# B&R Automation Studio project mappFramework (part 7)

#### HMIActions.st
```iecst
ACTION ReportFormat:

	// If the current format and the selected format do not match, disable the function block for a cycle and make the change
	IF HmiReport.Parameters.UseAdvancedFormat AND (HmiReport.Status.CurrentFormat = FORMAT_SIMPLE) THEN
		MpReportCoreSys.Enable := FALSE;
		MpReportCoreSys.MpLink := ADR(gMpLinkAdvancedReport);
		HmiReport.Parameters.Name := 'AdvancedReport';
		HmiReport.Status.CurrentFormat := FORMAT_ADVANCED;
	ELSIF NOT HmiReport.Parameters.UseAdvancedFormat AND (HmiReport.Status.CurrentFormat = FORMAT_ADVANCED) THEN
		MpReportCoreSys.Enable := FALSE;
		MpReportCoreSys.MpLink := ADR(gMpLinkSimpleReport);
		HmiReport.Parameters.Name := 'SimpleReport';
		HmiReport.Status.CurrentFormat := FORMAT_SIMPLE;
	ELSE
		MpReportCoreSys.Enable := TRUE;
	END_IF

END_ACTION

ACTION ReportFileExplorer:

	// Connections between the HMI structure and the report function block
	HmiReport.Status.Busy := MpReportCoreSys.CommandBusy;
	HmiReport.Status.Error := MpReportCoreSys.Error;
	MpReportCoreSys.Language := ADR(HmiReport.Parameters.SelectedLanguage);

	// Set or reset bits based on when a report can be created, deleted, and/or viewed.
	HmiReport.Status.CreateAllowed := NOT(MpReportCoreSys.CommandBusy);
	HmiReport.Status.ViewAllowed := (MpFileManagerUIConnect.File.List.Items[HmiReport.Status.SelectedIndex].ItemType = mpFILE_ITEM_TYPE_USER1);
	HmiReport.Status.DeleteAllowed := (MpFileManagerUIConnect.File.List.Items[HmiReport.Status.SelectedIndex].ItemType = mpFILE_ITEM_TYPE_USER1);

	// If the selected index on screen matches the index of a given file, mark that file as selected in the UIConnect structure
	FOR i := 0 TO ((SIZEOF(HmiReport.Status.FileNames)/SIZEOF(HmiReport.Status.FileNames[0])) - 1) DO
		IF (i = HmiReport.Status.SelectedIndex) AND NOT MpFileManagerUIConnect.File.List.Items[i].IsSelected THEN
			MpFileManagerUIConnect.File.List.Items[i].IsSelected := TRUE;
		ELSIF (i <> HmiReport.Status.SelectedIndex) AND MpFileManagerUIConnect.File.List.Items[i].IsSelected THEN
			MpFileManagerUIConnect.File.List.Items[i].IsSelected := FALSE;
		END_IF
	END_FOR

	// For every file, record its name, timestamp, size, and path
	FOR i := 0 TO ((SIZEOF(HmiReport.Status.FileNames)/SIZEOF(HmiReport.Status.FileNames[0])) - 1) DO
		HmiReport.Status.FileNames[i] := MpFileManagerUIConnect.File.List.Items[i].Name;
		HmiReport.Status.TimeStamps[i] := MpFileManagerUIConnect.File.List.Items[i].LastModified;

		IF MpFileManagerUIConnect.File.List.Items[i].Size <> 0 THEN
			HmiReport.Status.TimeStampsText[i] := DT_TO_STRING(MpFileManagerUIConnect.File.List.Items[i].LastModified);
			HmiReport.Status.TimeStampsText[i] := RIGHT(HmiReport.Status.TimeStampsText[i], 19);
		ELSE
			HmiReport.Status.TimeStampsText[i] := '';
		END_IF;

		HmiReport.Status.Size[i] := MpFileManagerUIConnect.File.List.Items[i].Size;
		// Concatonate strings to form the file path
		HmiReport.Status.TempFilePath[i] := '/FileDevice:';
		brsstrcat(ADR(HmiReport.Status.TempFilePath[i]),ADR(MpFileManagerUIConnect.DeviceList.DeviceNames[MpFileManagerUIConnect.DeviceList.SelectedIndex]));
		brsstrcat(ADR(HmiReport.Status.TempFilePath[i]),ADR('/'));
		brsstrcat(ADR(HmiReport.Status.TempFilePath[i]),ADR(HmiReport.Status.FileNames[i]));
		HmiReport.Status.FilePath[i] := HmiReport.Status.TempFilePath[i];
	END_FOR

	// Create a file path to be linked to the pdf viewer
	HmiReport.Parameters.PathOfReportToView := HmiReport.Status.FilePath[HmiReport.Status.SelectedIndex];

	// Add USB devices if available
	FOR i := 0 TO IDX_USB_DEV_LIST DO
		tempDeviceIndex := i + 1;
		IF gUSBAvailable[i] THEN
			MpFileManagerUIConnect.DeviceList.DeviceNames[tempDeviceIndex] := 'USB';
			brsitoa(i + 1, ADR(MpFileManagerUIConnect.DeviceList.DeviceNames[tempDeviceIndex]) + brsstrlen(ADR(MpFileManagerUIConnect.DeviceList.DeviceNames[tempDeviceIndex])));
		ELSE
			MpFileManagerUIConnect.DeviceList.DeviceNames[tempDeviceIndex] := '';
		END_IF
	END_FOR

	// Create array for the file device table
	IF ((MpFileManagerUIConnect.DeviceList.SelectedIndex <> HmiReport.Status.LastSelectedDeviceIndex) AND (MpFileManagerUIConnect.Status = mpFILE_UI_STATUS_IDLE)) THEN
		HmiReport.Status.LastSelectedDeviceIndex := MpFileManagerUIConnect.DeviceList.SelectedIndex;
		HmiReport.Status.LastSelectedIndex := HmiReport.Status.LastSelectedIndex + 1;
	END_IF

	// If more than 50 items exist, set the File OverMax flag (used for page up/down buttons)
	HmiReport.Status.FileOverMax := ItemCount > 50;

	// Set file device to selected
	MpReportCoreSys.DeviceName := ADR(MpFileManagerUIConnect.DeviceList.DeviceNames[MpFileManagerUIConnect.DeviceList.SelectedIndex]);

	// VC4
	IF HmiReport.Status.Error THEN
		HmiReport.Status.Layer.ReportCreate := USINT_TO_BOOL(HIDE);
	END_IF
	IF HmiReport.Status.DeleteAllowed THEN
		HmiReport.Status.DeleteButtonEnableStatus := USINT_TO_BOOL(HIDE);
	ELSE
		HmiReport.Status.DeleteButtonEnableStatus := USINT_TO_BOOL(DISPLAY);
	END_IF
	IF HmiReport.Status.FileOverMax THEN
		HmiReport.Status.PageUpDownVisibility := DISPLAY;
	ELSE
		HmiReport.Status.PageUpDownVisibility := HIDE;
	END_IF

	// Language assignments
	CASE HmiReport.Parameters.Language OF

		// English
		0:
			MpReportCoreSys.Language := ADR('en');
		// German
		1:
			MpReportCoreSys.Language := ADR('de');
		// Chinese
		2:
			MpReportCoreSys.Language := ADR('zh');

	END_CASE

END_ACTION
```

#### ReportMgr.st
```iecst
//***********************************************************************
// Copyright: B&R Industrial Automation GmbH
// Author: B&R Industrial Automation GmbH
// Created: Dec 1, 2022
// Description: Task for generating reports with VC4 front-end.
//***********************************************************************

PROGRAM _INIT

	// Create folder for this component on the user file device
	DirCreateReport(enable := TRUE, pDevice := ADR('mappReportFiles'), pName := ADR('/'));

	// Check if folder already exist and if so disabled the function block call
	IF DirCreateReport.status = fiERR_DIR_ALREADY_EXIST THEN
		DirCreateReport(enable := FALSE);
	END_IF

	// Initialize mapp function blocks
	MpReportCoreSys.Language := ADR('en');
	MpReportCoreSys.DeviceName := ADR('mappReportFiles');
	MpReportCoreSys.MpLink := ADR(gMpLinkSimpleReport);
	MpReportCoreSys.Name := ADR(HmiReport.Parameters.Name);
	HmiReport.Parameters.Name := 'SimpleReport';
	HmiReport.Parameters.SortType := 'NameAsc';
	MpReportCoreSys();

	MpFileManagerUIReport.MpLink := ADR(gMpLinkFileManagerUIReport);
	MpFileManagerUIReport.UIConnect := ADR(MpFileManagerUIConnect);
	MpFileManagerUIReport.UISetup.FileListSize := SIZEOF(MpFileManagerUIConnect.File.List.Items) / SIZEOF(MpFileManagerUIConnect.File.List.Items[0]);
	MpFileManagerUIReport.Enable := TRUE;
	MpFileManagerUIReport();

	// Fill an array to create example data for the example report
	TimeIndex := 0;
	FOR i:=0 TO ((SIZEOF(ReportExample.SimpleReport.OeeLine[0].TemperatureSample.TimeStamp)/SIZEOF(ReportExample.SimpleReport.OeeLine[0].TemperatureSample.TimeStamp[0])) - 1) DO
		ReportExample.SimpleReport.OeeLine[0].TemperatureSample.TimeStamp[i] := TimeIndex;
		ReportExample.SimpleReport.OeeLine[1].TemperatureSample.TimeStamp[i] := TimeIndex;
		ReportExample.SimpleReport.OeeLine[2].TemperatureSample.TimeStamp[i] := TimeIndex;
		ReportExample.AdvancedReport.OeeLine[0].TemperatureSample.TimeStamp[i] := TimeIndex;
		ReportExample.AdvancedReport.OeeLine[1].TemperatureSample.TimeStamp[i] := TimeIndex;
		ReportExample.AdvancedReport.OeeLine[2].TemperatureSample.TimeStamp[i] := TimeIndex;
		TimeIndex := TimeIndex + 15;
	END_FOR

	// Ficticious number to serve as an example in the report
	ReportExample.AdvancedReport.BatchNumber := 325454685;

END_PROGRAM

PROGRAM _CYCLIC

	// Once a report has been generated, clear the generate command
	IF MpReportCoreSys.CommandDone THEN
		MpFileManagerUIConnect.File.Refresh := TRUE;
		HmiReport.Commands.Generate := FALSE;
	END_IF

	// Call all cyclic actions
	ReportFormat;
	ReportFileExplorer;

	// Generate command
	MpReportCoreSys.Generate := HmiReport.Commands.Generate;
	MpReportCoreSys.Name := ADR(HmiReport.Parameters.Name);

	// Assign address references
	MpFileManagerUIReport.UIConnect := ADR(MpFileManagerUIConnect);
	MpFileManagerUIReport.MpLink := ADR(gMpLinkFileManagerUIReport);
	MpFileManagerUIReport.UIConnect := ADR(MpFileManagerUIConnect);

	// Call function blocks
	MpReportCoreSys();
	MpFileManagerUIReport();

END_PROGRAM

PROGRAM _EXIT

	// Disable the function blocks to unlink the MpLinks
	MpReportCoreSys.Enable := FALSE;
	MpFileManagerUIReport.Enable := FALSE;

	// Call function blocks
	MpReportCoreSys();
	MpFileManagerUIReport();

END_PROGRAM
```

### mappFrameworkVC4.var - not listed in the package file held
```iecst
(*Constants*)
VAR CONSTANT
	DISPLAY : USINT := 0; (*VC4 visibility control*)
	HIDE : USINT := 1; (*VC4 visibility control*)
	OPERATION_ACTIVATED : USINT := 1; (*VC4 access control*)
	OPERATION_DEACTIVATED : USINT := 0; (*VC4 access control*)
	LOCK : USINT := 0; (*VC4 lock control*)
	UNLOCK : USINT := 1; (*VC4 unlock control*)
END_VAR
```

### Program Logical/Infrastructure/VC4/PackML/PackMLMgr (IEC)

#### PackMLMgr.st - Init, cyclic, exit code
```iecst
//***********************************************************************
// Copyright: B&R Industrial Automation GmbH
// Author: B&R Industrial Automation GmbH
// Created: June 1, 2023
// Description: Task for handling PackML control with VC4 front-end.
//***********************************************************************

PROGRAM _INIT

	// NOTE: For VC4 implementations, the MpPackMLCore must be configured in "standalone" mode.
	// For additional information, see "Required Modifications" in AS Mapp Framework Help.

	// Create folder for this component on the user file device
	DirCreatePackML(enable := TRUE, pDevice := ADR('mappPackMLFiles'), pName := ADR('/'));

	// Check if folder already exist and if so disabled the function block call
	IF DirCreatePackML.status = fiERR_DIR_ALREADY_EXIST THEN
		DirCreatePackML(enable := FALSE);
	END_IF

	// Initialize mapp function blocks
	MpPackMLCoreMain.MpLink := ADR(gMpLinkPackMLCore);
	MpPackMLCoreMain.Enable := TRUE;
	MpPackMLCoreMain();

	MpPackMLModeMain.MpLink := ADR(gMpLinkPackMLCore);
	MpPackMLModeMain.Enable := TRUE;
	MpPackMLModeMain.ModeID := 1;
	MpPackMLModeMain();

	MpPackMLBasicUIMain.MpLink := ADR(gMpLinkPackMLCore);
	MpPackMLBasicUIMain.Enable := TRUE;
	MpPackMLBasicUIMain.UIConnect := ADR(MpPackMLBasicUIConnect);
	MpPackMLBasicUIMain();

	MpPackMLStatisticsUIMain.MpLink := ADR(gMpLinkPackMLCore);
	MpPackMLStatisticsUIMain.Enable := TRUE;
	MpPackMLStatisticsUIMain.UIConnect := ADR(MpPackMLStatisticsUIConnect);
	MpPackMLStatisticsUIMain();

	// Assign Production mode as selected Index since it's the start mode and preselected
	MpPackMLBasicUIConnect.ModeControl.SelectedIndex := 1;

END_PROGRAM

PROGRAM _CYCLIC

	// Call all cyclic actions
	StateMachine;

	// Assign MpLinks & UIConnects
	MpPackMLCoreMain.MpLink := ADR(gMpLinkPackMLCore);
	MpPackMLModeMain.MpLink := ADR(gMpLinkPackMLCore);
	MpPackMLBasicUIMain.MpLink := ADR(gMpLinkPackMLCore);
	MpPackMLStatisticsUIMain.MpLink := ADR(gMpLinkPackMLCore);

	// Call function blocks
	MpPackMLCoreMain();
	MpPackMLModeMain();
	MpPackMLBasicUIMain();
	MpPackMLStatisticsUIMain();

END_PROGRAM

PROGRAM _EXIT

	// Disable the function blocks to unlink the MpLinks
	MpPackMLCoreMain.Enable := FALSE;
	MpPackMLModeMain.Enable := FALSE;
	MpPackMLBasicUIMain.Enable := FALSE;
	MpPackMLStatisticsUIMain.Enable := TRUE;

	// Call function blocks
	MpPackMLCoreMain();
	MpPackMLModeMain();
	MpPackMLBasicUIMain();
	MpPackMLStatisticsUIMain();

END_PROGRAM
```

#### PackMLMgr.var - Local variables
```iecst
(*Function Blocks*)
VAR
	DirCreatePackML : DirCreate; (*DirCreate instance*)
	MpPackMLCoreMain : MpPackMLCore;
	MpPackMLModeMain : MpPackMLMode;
	MpPackMLBasicUIMain : MpPackMLBasicUI;
	MpPackMLStatisticsUIMain : MpPackMLStatisticsUI;
END_VAR
(*Constants*)
(*Structure Types*)
VAR
	MpPackMLBasicUIConnect : MpPackMLBasicUIConnectType;
END_VAR
(*Variables*)
VAR
	MpPackMLStatisticsUIConnect : MpPackMLStatisticsUIConnectType;
END_VAR
```

#### StateMachine.st
```iecst
ACTION StateMachine:

	CASE MpPackMLCoreMain.StateCurrent OF

		mpPACKML_STATE_STOPPED:

			// Add STOPPED actions here
			MpPackMLModeMain.StateComplete := FALSE;

		mpPACKML_STATE_STARTING:

			// Add STARTING actions here
			MpPackMLModeMain.StateComplete := TRUE;

		mpPACKML_STATE_IDLE:

			// Add IDLE actions here
			MpPackMLModeMain.StateComplete := FALSE;

		mpPACKML_STATE_SUSPENDING:

			// Add SUSPENDING actions here
			MpPackMLModeMain.StateComplete := TRUE;

		mpPACKML_STATE_SUSPENDED:

			// Add SUSPENDED actions here
			MpPackMLModeMain.StateComplete := FALSE;

		mpPACKML_STATE_UNSUSPENDING:

			// Add UNSUSPENDING actions here
			MpPackMLModeMain.StateComplete := TRUE;

		mpPACKML_STATE_EXECUTE:

			// Add EXECUTE actions here
			MpPackMLModeMain.StateComplete := FALSE;

		mpPACKML_STATE_STOPPING:

			// Add STOPPING actions here
			MpPackMLModeMain.StateComplete := TRUE;

		mpPACKML_STATE_ABORTING:

			// Add ABORTING actions here
			MpPackMLModeMain.StateComplete := TRUE;

		mpPACKML_STATE_ABORTED:

			// Add ABORTED actions here
			MpPackMLModeMain.StateComplete := FALSE;

		mpPACKML_STATE_HOLDING:

			// Add HOLDING actions here
			MpPackMLModeMain.StateComplete := TRUE;

		mpPACKML_STATE_HELD:

			// Add HELD actions here
			MpPackMLModeMain.StateComplete := FALSE;

		mpPACKML_STATE_UNHOLDING:

			// Add UNHOLDING actions here
			MpPackMLModeMain.StateComplete := TRUE;

		mpPACKML_STATE_COMPLETING:

			// Add COMPLETING actions here
			MpPackMLModeMain.StateComplete := TRUE;

			// NOTE: To allow the state machine to move forward, the StateComplete command has been connected
			// to the HMI button. The user should change this to set StateComplete to TRUE upon COMPLETING actions.

		mpPACKML_STATE_COMPLETE:

			// Add COMPLETE actions here
			MpPackMLModeMain.StateComplete := FALSE;

		mpPACKML_STATE_RESETTING:

			// Add RESETTING actions here
			MpPackMLModeMain.StateComplete := TRUE;

		mpPACKML_STATE_CLEARING:

			// Add CLEARING actions here
			MpPackMLModeMain.StateComplete := TRUE;

		mpPACKML_STATE_UNDEFINED:

			// Add UNDEFINED actions here
			MpPackMLModeMain.Activate := TRUE;

		mpPACKML_STATE_DEACTIVATING:

			// Add DEACTIVATING actions here

		mpPACKML_STATE_DEACTIVATED:

			// Add DEACTIVATED actions here

		mpPACKML_STATE_ACTIVATING:

			// Add ACTIVATING actions here

			MpPackMLModeMain.StateComplete := TRUE;

	END_CASE

END_ACTION
```

#### HMIActions.st - not listed in the package file held
```iecst
ACTION VC4_Cyclic:

	IF HmiPackML.Status.LastState <> MpPackMLMode_0.StateCurrent THEN

		// Reset all commands on each state change
		MpPackMLBasicUIConnect.StateControl.Abort := MpPackMLMode_0.Abort := FALSE;
		MpPackMLBasicUIConnect.StateControl.Clear := MpPackMLMode_0.Clear := FALSE;
		MpPackMLBasicUIConnect.StateControl.Hold := MpPackMLMode_0.Hold := FALSE;
		MpPackMLBasicUIConnect.StateControl.Reset := MpPackMLMode_0.Reset := FALSE;
		MpPackMLBasicUIConnect.StateControl.Start := MpPackMLMode_0.Start := FALSE;
		MpPackMLBasicUIConnect.StateControl.StateComplete := MpPackMLMode_0.StateComplete := FALSE;
		MpPackMLBasicUIConnect.StateControl.Stop := MpPackMLMode_0.Stop := FALSE;
		MpPackMLBasicUIConnect.StateControl.Suspend := MpPackMLMode_0.Suspend := FALSE;
		MpPackMLBasicUIConnect.StateControl.Unhold := MpPackMLMode_0.Unhold := FALSE;
		MpPackMLBasicUIConnect.StateControl.Unsuspend := MpPackMLMode_0.Unsuspend := FALSE;

		// Reset all ColorIndexes on each state change
		MpPackMLBasicUIConnect.StateControl.ColorIndex.Stopped := 0;
		MpPackMLBasicUIConnect.StateControl.ColorIndex.Stopping := 0;
		MpPackMLBasicUIConnect.StateControl.ColorIndex.Clearing := 0;
		MpPackMLBasicUIConnect.StateControl.ColorIndex.Aborted := 0;
		MpPackMLBasicUIConnect.StateControl.ColorIndex.Aborting := 0;
		MpPackMLBasicUIConnect.StateControl.ColorIndex.Resetting := 0;
		MpPackMLBasicUIConnect.StateControl.ColorIndex.Unsuspending := 0;
		MpPackMLBasicUIConnect.StateControl.ColorIndex.Suspended := 0;
		MpPackMLBasicUIConnect.StateControl.ColorIndex.Suspending := 0;
		MpPackMLBasicUIConnect.StateControl.ColorIndex.Idle := 0;
		MpPackMLBasicUIConnect.StateControl.ColorIndex.Starting := 0;
		MpPackMLBasicUIConnect.StateControl.ColorIndex.Execute := 0;
		MpPackMLBasicUIConnect.StateControl.ColorIndex.Completing := 0;
		MpPackMLBasicUIConnect.StateControl.ColorIndex.Complete := 0;
		MpPackMLBasicUIConnect.StateControl.ColorIndex.Unholding := 0;
		MpPackMLBasicUIConnect.StateControl.ColorIndex.Held := 0;
		MpPackMLBasicUIConnect.StateControl.ColorIndex.Holding := 0;

		HmiPackML.Status.LastState := MpPackMLMode_0.StateCurrent;

	END_IF

	// Connect UIConnect Commands to function block
	MpPackMLMode_0.Abort := MpPackMLBasicUIConnect.StateControl.Abort;
	MpPackMLMode_0.Stop := MpPackMLBasicUIConnect.StateControl.Stop;

	MpPackMLBasicUIConnect.ModeCurrent := MpPackMLMode_0.ModeID;
	MpPackMLBasicUIConnect.StateCurrent := MpPackMLMode_0.StateCurrent;

END_ACTION
```

#### StateMachine_Main.st - not listed in the package file held
```iecst
ACTION StateMachine_Main:

	CASE MpPackMLCore_0.StateCurrent OF

		mpPACKML_STATE_STOPPED:

			// Add STOPPED actions here
			MpPackMLMode_0.StateComplete := FALSE;

		mpPACKML_STATE_STARTING:

			// Add STARTING actions here
			MpPackMLMode_0.StateComplete := TRUE;

		mpPACKML_STATE_IDLE:

			// Add IDLE actions here
			MpPackMLMode_0.StateComplete := FALSE;

		mpPACKML_STATE_SUSPENDING:

			// Add SUSPENDING actions here
			MpPackMLMode_0.StateComplete := TRUE;

		mpPACKML_STATE_SUSPENDED:

			// Add SUSPENDED actions here
			MpPackMLMode_0.StateComplete := FALSE;

		mpPACKML_STATE_UNSUSPENDING:

			// Add UNSUSPENDING actions here
			MpPackMLMode_0.StateComplete := TRUE;

		mpPACKML_STATE_EXECUTE:

			// Add EXECUTE actions here
			MpPackMLMode_0.StateComplete := FALSE;

		mpPACKML_STATE_STOPPING:

			// Add STOPPING actions here
			MpPackMLMode_0.StateComplete := TRUE;

		mpPACKML_STATE_ABORTING:

			// Add ABORTING actions here
			MpPackMLMode_0.StateComplete := TRUE;

		mpPACKML_STATE_ABORTED:

			// Add ABORTED actions here
			MpPackMLMode_0.StateComplete := FALSE;

		mpPACKML_STATE_HOLDING:

			// Add HOLDING actions here
			MpPackMLMode_0.StateComplete := TRUE;

		mpPACKML_STATE_HELD:

			// Add HELD actions here
			MpPackMLMode_0.StateComplete := FALSE;

		mpPACKML_STATE_UNHOLDING:

			// Add UNHOLDING actions here
			MpPackMLMode_0.StateComplete := TRUE;

		mpPACKML_STATE_COMPLETING:

			// Add COMPLETING actions here
			MpPackMLMode_0.StateComplete := TRUE;

			// NOTE: To allow the state machine to move forward, the StateComplete command has been connected
			// to the HMI button. The user should change this to set StateComplete to TRUE upon COMPLETING actions.

		mpPACKML_STATE_COMPLETE:

			// Add COMPLETE actions here
			MpPackMLMode_0.StateComplete := FALSE;

		mpPACKML_STATE_RESETTING:

			// Add RESETTING actions here
			MpPackMLMode_0.StateComplete := TRUE;

		mpPACKML_STATE_CLEARING:

			// Add CLEARING actions here
			MpPackMLMode_0.StateComplete := TRUE;

		mpPACKML_STATE_UNDEFINED:

			// Add UNDEFINED actions here
			MpPackMLMode_0.Activate := TRUE;

		mpPACKML_STATE_DEACTIVATING:

			// Add DEACTIVATING actions here

		mpPACKML_STATE_DEACTIVATED:

			// Add DEACTIVATED actions here

		mpPACKML_STATE_ACTIVATING:

			// Add ACTIVATING actions here

			MpPackMLMode_0.StateComplete := TRUE;

	END_CASE

END_ACTION
```

### Program Logical/Infrastructure/PackML/PackMLMgr (IEC) - Pack ML Manager

#### PackMLMgr.st - Init, cyclic, exit code
```iecst
//***********************************************************************
// Copyright: B&R Industrial Automation GmbH
// Author: B&R Industrial Automation GmbH
// Created: June 1, 2023
// Description: Task for handling PackML control.
//***********************************************************************

PROGRAM _INIT

	// Create folder for this component on the user file device
	DirCreatePackML(enable := TRUE, pDevice := ADR('mappPackMLFiles'), pName := ADR('/'));

	// Check if folder already exist and if so disabled the function block call
	IF DirCreatePackML.status = fiERR_DIR_ALREADY_EXIST THEN
		DirCreatePackML(enable := FALSE);
	END_IF

	// Initialize mapp function blocks
	MpPackMLModuleMain.Parameters := ADR(MpPackMLModuleParMain);
	MpPackMLModuleMain.MpLink := ADR(gMpPackMLModuleMain);
	MpPackMLModuleMain.Enable := TRUE;
	MpPackMLModuleMain();

	//PackML Mode Initializations
	StateInitialize;

	// Initialize startup mode - Automatic Mode
	HmiPackML.Commands.Mode := 1;

END_PROGRAM

PROGRAM _CYCLIC

	// Call all cyclic actions
	StateMachine;
	HmiActions;

	// Assign MpLinks & UIConnects
	MpPackMLModuleMain.Parameters := ADR(MpPackMLModuleParMain);
	MpPackMLModuleMain.MpLink := ADR(gMpPackMLModuleMain);

	// Call function blocks
	MpPackMLModuleMain();

END_PROGRAM

PROGRAM _EXIT

	// Disable the function blocks to unlink the MpLinks
	MpPackMLModuleMain.Enable := FALSE;

	// Call function blocks
	MpPackMLModuleMain();

END_PROGRAM
```

#### PackMLMgr.typ - Local data types
```iecst
(*Structure types*)

TYPE
	PackMLHmiInterfaceType : 	STRUCT  (*Structure to hold commands, parameters and status from the HMI*)
		Commands : PackMLCommandsType;
		Parameters : PackMLParametersType;
		Status : PackMLStatusType;
		Activate : BOOL;
	END_STRUCT;
	PackMLCommandsType : 	STRUCT  (*Structure to hold the commands from the HMI*)
		Reset : BOOL;
		Start : BOOL;
		Stop : BOOL;
		Hold : BOOL;
		Unhold : BOOL;
		Suspend : BOOL;
		Unsuspend : BOOL;
		Abort : BOOL;
		Clear : BOOL;
		Complete : BOOL;
		Mode : DINT;
	END_STRUCT;
	PackMLParametersType : 	STRUCT  (*Structure to hold the parameters for the HMI*)
		Par : USINT;
		StateEnabled : PackMLStateEnabledType;
	END_STRUCT;
	PackMLStatusType : 	STRUCT  (*Structure to hold status information from the mapp View HMI*)
		StateCurrent : STRING[20];
		ModeCurrent : STRING[50];
		DownTimeReason : STRING[255];
		PackMLStateModel : STRING[100000];
		PackMLState : MpPackMLStateEnum;
	END_STRUCT;
	PackMLStateEnabledType : 	STRUCT  (*Structure to hold state availability definition*)
		Clearing : BOOL; (*Statistic information for Clearing state*)
		Stopped : BOOL; (*Statistic information for Stopped state*)
		Starting : BOOL; (*Statistic information for Starting state*)
		Idle : BOOL; (*Statistic information for Idle state*)
		Suspended : BOOL; (*Statistic information for Suspended state*)
		Execute : BOOL; (*Statistic information for Execute state*)
		Stopping : BOOL; (*Statistic information for Stopping state*)
		Aborting : BOOL; (*Statistic information for Aborting state*)
		Aborted : BOOL; (*Statistic information for Aborted state*)
		Holding : BOOL; (*Statistic information for Holding state*)
		Held : BOOL; (*Statistic information for Held state*)
		Unholding : BOOL; (*Statistic information for Unholding state*)
		Suspending : BOOL; (*Statistic information for Suspending state*)
		Unsuspending : BOOL; (*Statistic information for Unsuspending state*)
		Resetting : BOOL; (*Statistic information for Resetting state*)
		Completing : BOOL; (*Statistic information for Completing state*)
		Complete : BOOL; (*Statistic information for Complete state*)
	END_STRUCT;
END_TYPE

(*Enumerations*)
```

#### PackMLMgr.var - Local variables
```iecst
(*Function Blocks*)
VAR
	DirCreatePackML : DirCreate; (*DirCreate instance*)
	MpPackMLModuleMain : MpPackMLModule; (*PackMLModule instance*)
	MpPackMLModuleParMain : MpPackMLModuleParType; (*PackMLModule Parameter instance*)
	StateBlinkTimer : TON; (*Timer to control state blinking action*)
END_VAR
(*Constants*)
(*Structure Types*)
VAR
	Manual : PackMLStateEnabledType; (*State active / inactive control*)
	Maintenance : PackMLStateEnabledType; (*State active / inactive control*)
	AutomaticMode : PackMLStateEnabledType; (*State active / inactive control*)
	HmiPackML : PackMLHmiInterfaceType; (*HMI interface structure*)
END_VAR
(*Variables*)
```

#### HMIActions.st - Supporting code for the HMI interface
```iecst
ACTION HmiActions:

	// Connect HMIPackML Commands to function block
	MpPackMLModuleMain.Command.Abort := HmiPackML.Commands.Abort;
	MpPackMLModuleMain.Command.Clear := HmiPackML.Commands.Clear;
	MpPackMLModuleMain.Command.Hold := HmiPackML.Commands.Hold;
	MpPackMLModuleMain.Command.Reset := HmiPackML.Commands.Reset;
	MpPackMLModuleMain.Command.Start := HmiPackML.Commands.Start;
	MpPackMLModuleMain.Command.Stop := HmiPackML.Commands.Stop;
	MpPackMLModuleMain.Command.Suspend := HmiPackML.Commands.Suspend;
	MpPackMLModuleMain.Command.Unhold := HmiPackML.Commands.Unhold;
	MpPackMLModuleMain.Command.Unsuspend := HmiPackML.Commands.Unsuspend;

	// Allow user to command StateComplete only while machine is in state execute
	IF MpPackMLModuleMain.StateCurrent = mpPACKML_STATE_EXECUTE THEN
		MpPackMLModuleMain.Command.StateComplete := HmiPackML.Commands.Complete;
	END_IF

	// Assign mode configuration based on active mode
	CASE MpPackMLModuleMain.ModeID OF
		1:
			HmiPackML.Parameters.StateEnabled := AutomaticMode;
		2:
			HmiPackML.Parameters.StateEnabled := Maintenance;
		3:
			HmiPackML.Parameters.StateEnabled := Manual;
	END_CASE

	// control state machine active state blinking
	CASE HmiPackML.Status.PackMLState OF

		0:	// Build the intital string to setup enabled states and reduce the opacity to 50% for inactive states

			PackMLBaseModel(HmiPackML.Parameters.StateEnabled,ADR(HmiPackML.Status.PackMLStateModel));

			//start timer before transitioning to the current state which turns the opacity to 100% creating a blinking effect
			StateBlinkTimer.IN := TRUE;
			IF StateBlinkTimer.Q THEN
				HmiPackML.Status.PackMLState := MpPackMLModuleMain.StateCurrent;
				StateBlinkTimer.IN := FALSE;
			END_IF

		mpPACKML_STATE_CLEARING..mpPACKML_STATE_COMPLETE:

			StateBlinkTimer.IN := TRUE;
			IF StateBlinkTimer.Q THEN
				HmiPackML.Status.PackMLState := 0;
				StateBlinkTimer.IN := FALSE;
			END_IF

		ELSE	//if the state does't exist because of the synchronized mode use just go back to state 0
			HmiPackML.Status.PackMLState := 0;
	END_CASE

	// timer function block call
	StateBlinkTimer(PT := t#1s);

	// copy status info to HMI structure
	HmiPackML.Status.StateCurrent := MpPackMLModuleMain.Info.StateCurrent;
	HmiPackML.Status.ModeCurrent := MpPackMLModuleMain.Info.ModeCurrent;

END_ACTION
```

#### StateMachine.st - Main state machine logic
```iecst
ACTION StateMachine:

	// Check active state and change mode if allowed
	IF MpPackMLModeChangeIsAllowed(gMpLinkPackMLCore,HmiPackML.Commands.Mode) = 0 THEN
		MpPackMLChangeMode(gMpLinkPackMLCore,HmiPackML.Commands.Mode);
	END_IF

	CASE MpPackMLModuleMain.StateCurrent OF

		mpPACKML_STATE_STOPPED:

			// Add STOPPED actions here

		mpPACKML_STATE_STARTING:

			// Add STARTING actions here

			MpPackMLModuleMain.Command.StateComplete := TRUE;

		mpPACKML_STATE_IDLE:

			// Add IDLE actions here

		mpPACKML_STATE_SUSPENDING:

			// Add SUSPENDING actions here

			MpPackMLModuleMain.Command.StateComplete := TRUE;

		mpPACKML_STATE_SUSPENDED:

			// Add SUSPENDED actions here

		mpPACKML_STATE_UNSUSPENDING:

			// Add UNSUSPENDING actions here

			MpPackMLModuleMain.Command.StateComplete := TRUE;

		mpPACKML_STATE_EXECUTE:

			// Add EXECUTE actions here

		mpPACKML_STATE_STOPPING:

			// Add STOPPING actions here

			MpPackMLModuleMain.Command.StateComplete := TRUE;

		mpPACKML_STATE_ABORTING:

			// Add ABORTING actions here

			MpPackMLModuleMain.Command.StateComplete := TRUE;

		mpPACKML_STATE_ABORTED:

			// Add ABORTED actions here

		mpPACKML_STATE_HOLDING:

			// Add HOLDING actions here

			MpPackMLModuleMain.Command.StateComplete := TRUE;

		mpPACKML_STATE_HELD:

			// Add HELD actions here

		mpPACKML_STATE_UNHOLDING:

			// Add UNHOLDING actions here

			MpPackMLModuleMain.Command.StateComplete := TRUE;

		mpPACKML_STATE_COMPLETING:

			// Add COMPLETING actions here

			// NOTE: once COMPLETING actions that take more than one cyclic have been added, the below line
			// should be removed and replaced by the following line.
			MpPackMLModuleMain.Command.StateComplete := NOT MpPackMLModuleMain.Command.StateComplete;
			// MpPackMLModuleMain.Command.StateComplete := TRUE;

		mpPACKML_STATE_COMPLETE:

			// Add COMPLETE actions here

		mpPACKML_STATE_RESETTING:

			// Add RESETTING actions here

			MpPackMLModuleMain.Command.StateComplete := TRUE;

		mpPACKML_STATE_CLEARING:

			// Add CLEARING actions here

			MpPackMLModuleMain.Command.StateComplete := TRUE;

		mpPACKML_STATE_DEACTIVATING:

			// Add DEACTIVATING actions here

		mpPACKML_STATE_DEACTIVATED:

			// Add DEACTIVATED actions here

		mpPACKML_STATE_ACTIVATING:

			// Add ACTIVATING actions here

			MpPackMLModuleMain.Command.StateComplete := TRUE;

	END_CASE

END_ACTION
```

#### LocalFunctions.fun - Declaration for local helper functions
```iecst
{REDUND_ERROR} FUNCTION PackMLBaseModel : BOOL (* *) (*$GROUP=User,$CAT=User,$GROUPICON=User.png,$CATICON=User.png*)
	VAR_INPUT
		StateEnabled : PackMLStateEnabledType;
		BaseLayout : REFERENCE TO STRING[100000];
	END_VAR
	VAR
		stringPart : STRING[79];
	END_VAR
END_FUNCTION
```

#### PackMLBaseModel.st - Function to control the paper widget transform string
```iecst
FUNCTION PackMLBaseModel

			BaseLayout := '';
			brsstrcat(ADR(BaseLayout),ADR('['));

			IF StateEnabled.Clearing THEN
				stringPart := '{"select":"#Clearing","style":"fill:1;fill-opacity:1"}';
			ELSE
				stringPart := '{"select":"#Clearing","style":"fill:0;fill-opacity:0.5"}';
			END_IF

			brsstrcat(ADR(BaseLayout),ADR(stringPart));
			brsstrcat(ADR(BaseLayout),ADR(','));

			stringPart := '{"select":"#Stopped","style":"fill:2;fill-opacity:1"}';

			brsstrcat(ADR(BaseLayout),ADR(stringPart));
			brsstrcat(ADR(BaseLayout),ADR(','));

			IF StateEnabled.Starting THEN
				stringPart := '{"select":"#Starting","style":"fill:1;fill-opacity:1"}';
			ELSE
				stringPart := '{"select":"#Starting","style":"fill:0;fill-opacity:0.5"}';
			END_IF

			brsstrcat(ADR(BaseLayout),ADR(stringPart));
			brsstrcat(ADR(BaseLayout),ADR(','));

			stringPart := '{"select":"#Idle","style":"fill:2;fill-opacity:1"}';

			brsstrcat(ADR(BaseLayout),ADR(stringPart));
			brsstrcat(ADR(BaseLayout),ADR(','));

			IF StateEnabled.Suspended THEN
				stringPart := '{"select":"#Suspended","style":"fill:2;fill-opacity:1"}';
			ELSE
				stringPart := '{"select":"#Suspended","style":"fill:0;fill-opacity:0.5"}';
			END_IF

			brsstrcat(ADR(BaseLayout),ADR(stringPart));
			brsstrcat(ADR(BaseLayout),ADR(','));

			stringPart := '{"select":"#Execute","style":"fill:4;fill-opacity:1"}';

			brsstrcat(ADR(BaseLayout),ADR(stringPart));
			brsstrcat(ADR(BaseLayout),ADR(','));

			IF StateEnabled.Stopping THEN
				stringPart := '{"select":"#Stopping","style":"fill:1;fill-opacity:1"}';
			ELSE
				stringPart := '{"select":"#Stopping","style":"fill:0;fill-opacity:0.5"}';
			END_IF

			brsstrcat(ADR(BaseLayout),ADR(stringPart));
			brsstrcat(ADR(BaseLayout),ADR(','));

			IF StateEnabled.Aborting THEN
				stringPart := '{"select":"#Aborting","style":"fill:1;fill-opacity:1"}';
			ELSE
				stringPart := '{"select":"#Aborting","style":"fill:0;fill-opacity:0.5"}';
			END_IF

			brsstrcat(ADR(BaseLayout),ADR(stringPart));
			brsstrcat(ADR(BaseLayout),ADR(','));

			stringPart := '{"select":"#Aborted","style":"fill:2;fill-opacity:1"}';

			brsstrcat(ADR(BaseLayout),ADR(stringPart));
			brsstrcat(ADR(BaseLayout),ADR(','));

			IF StateEnabled.Holding THEN
				stringPart := '{"select":"#Holding","style":"fill:1;fill-opacity:1"}';
			ELSE
				stringPart := '{"select":"#Holding","style":"fill:0;fill-opacity:0.5"}';
			END_IF

			brsstrcat(ADR(BaseLayout),ADR(stringPart));
			brsstrcat(ADR(BaseLayout),ADR(','));

			IF StateEnabled.Held THEN
				stringPart := '{"select":"#Held","style":"fill:2;fill-opacity:1"}';
			ELSE
				stringPart := '{"select":"#Held","style":"fill:0;fill-opacity:0.5"}';
			END_IF

			brsstrcat(ADR(BaseLayout),ADR(stringPart));
			brsstrcat(ADR(BaseLayout),ADR(','));

			IF StateEnabled.Unholding THEN
				stringPart := '{"select":"#Unholding","style":"fill:1;fill-opacity:1"}';
			ELSE
				stringPart := '{"select":"#Unholding","style":"fill:0;fill-opacity:0.5"}';
			END_IF

			brsstrcat(ADR(BaseLayout),ADR(stringPart));
			brsstrcat(ADR(BaseLayout),ADR(','));

			IF StateEnabled.Suspending THEN
				stringPart := '{"select":"#Suspending","style":"fill:1;fill-opacity:1"}';
			ELSE
				stringPart := '{"select":"#Suspending","style":"fill:0;fill-opacity:0.5"}';
			END_IF

			brsstrcat(ADR(BaseLayout),ADR(stringPart));
			brsstrcat(ADR(BaseLayout),ADR(','));

			IF StateEnabled.Unsuspending THEN
				stringPart := '{"select":"#Unsuspending","style":"fill:1;fill-opacity:1"}';
			ELSE
				stringPart := '{"select":"#Unsuspending","style":"fill:0;fill-opacity:0.5"}';
			END_IF

			brsstrcat(ADR(BaseLayout),ADR(stringPart));
			brsstrcat(ADR(BaseLayout),ADR(','));

			IF StateEnabled.Resetting THEN
				stringPart := '{"select":"#Resetting","style":"fill:1;fill-opacity:1"}';
			ELSE
				stringPart := '{"select":"#Resetting","style":"fill:0;fill-opacity:0.5"}';
			END_IF

			brsstrcat(ADR(BaseLayout),ADR(stringPart));
			brsstrcat(ADR(BaseLayout),ADR(','));

			IF StateEnabled.Completing THEN
				stringPart := '{"select":"#Completing","style":"fill:1;fill-opacity:1"}';
			ELSE
				stringPart := '{"select":"#Completing","style":"fill:0;fill-opacity:0.5"}';
			END_IF

			brsstrcat(ADR(BaseLayout),ADR(stringPart));
			brsstrcat(ADR(BaseLayout),ADR(','));

			IF StateEnabled.Complete THEN
				stringPart := '{"select":"#Complete","style":"fill:2;fill-opacity:1"}';
			ELSE
				stringPart := '{"select":"#Complete","style":"fill:0;fill-opacity:0.5"}';
			END_IF

			brsstrcat(ADR(BaseLayout),ADR(stringPart));
			brsstrcat(ADR(BaseLayout),ADR(']'));

			PackMLBaseModel := TRUE;

END_FUNCTION
```

#### StateInitialize.st
```iecst
ACTION StateInitialize:

	//Initialize the PackML framework

	Manual.Clearing:=FALSE;
	Manual.Stopped:=TRUE;
	Manual.Starting:=TRUE;
	Manual.Idle:=TRUE;
	Manual.Suspended:=FALSE;
	Manual.Execute:=TRUE;
	Manual.Stopping:=TRUE;
	Manual.Aborting:=TRUE;
	Manual.Aborted:=TRUE;
	Manual.Holding:=FALSE;
	Manual.Held:=FALSE;
	Manual.Unholding:=FALSE;
	Manual.Suspending:=FALSE;
	Manual.Unsuspending:=FALSE;
	Manual.Resetting:=TRUE;
	Manual.Completing:=FALSE;
	Manual.Complete:=FALSE;

	Maintenance.Clearing:=TRUE;
	Maintenance.Stopped:=TRUE;
	Maintenance.Starting:=TRUE;
	Maintenance.Idle:=TRUE;
	Maintenance.Suspended:=FALSE;
	Maintenance.Execute:=TRUE;
	Maintenance.Stopping:=TRUE;
	Maintenance.Aborting:=TRUE;
	Maintenance.Aborted:=TRUE;
	Maintenance.Holding:=TRUE;
	Maintenance.Held:=TRUE;
	Maintenance.Unholding:=TRUE;
	Maintenance.Suspending:=FALSE;
	Maintenance.Unsuspending:=FALSE;
	Maintenance.Resetting:=TRUE;
	Maintenance.Completing:=FALSE;
	Maintenance.Complete:=FALSE;

	AutomaticMode.Clearing:=TRUE;
	AutomaticMode.Stopped:=TRUE;
	AutomaticMode.Starting:=TRUE;
	AutomaticMode.Idle:=TRUE;
	AutomaticMode.Suspended:=TRUE;
	AutomaticMode.Execute:=TRUE;
	AutomaticMode.Stopping:=TRUE;
	AutomaticMode.Aborting:=TRUE;
	AutomaticMode.Aborted:=TRUE;
	AutomaticMode.Holding:=TRUE;
	AutomaticMode.Held:=TRUE;
	AutomaticMode.Unholding:=TRUE;
	AutomaticMode.Suspending:=TRUE;
	AutomaticMode.Unsuspending:=TRUE;
	AutomaticMode.Resetting:=TRUE;
	AutomaticMode.Completing:=TRUE;
	AutomaticMode.Complete:=TRUE;

	HmiPackML.Parameters.StateEnabled.Clearing:=TRUE;
	HmiPackML.Parameters.StateEnabled.Stopped:=TRUE;
	HmiPackML.Parameters.StateEnabled.Starting:=TRUE;
	HmiPackML.Parameters.StateEnabled.Idle:=TRUE;
	HmiPackML.Parameters.StateEnabled.Suspended:=TRUE;
	HmiPackML.Parameters.StateEnabled.Execute:=TRUE;
	HmiPackML.Parameters.StateEnabled.Stopping:=TRUE;
	HmiPackML.Parameters.StateEnabled.Aborting:=TRUE;
	HmiPackML.Parameters.StateEnabled.Aborted:=TRUE;
	HmiPackML.Parameters.StateEnabled.Holding:=TRUE;
	HmiPackML.Parameters.StateEnabled.Held:=TRUE;
	HmiPackML.Parameters.StateEnabled.Unholding:=TRUE;
	HmiPackML.Parameters.StateEnabled.Suspending:=TRUE;
	HmiPackML.Parameters.StateEnabled.Unsuspending:=TRUE;
	HmiPackML.Parameters.StateEnabled.Resetting:=TRUE;
	HmiPackML.Parameters.StateEnabled.Completing:=TRUE;
	HmiPackML.Parameters.StateEnabled.Complete:=TRUE;

END_ACTION
```

#### StateMachine_Main.st - not listed in the package file held
```iecst
ACTION StateMachine_Main:

	// Check active state and change mode if allowed
	IF MpPackMLModeChangeIsAllowed(gMpLinkPackMLCore,HmiPackML.Commands.Mode) = 0 THEN
		MpPackMLChangeMode(gMpLinkPackMLCore,HmiPackML.Commands.Mode);
	END_IF

	CASE MpPackMLModule_Main.StateCurrent OF

		mpPACKML_STATE_STOPPED:

			// Add STOPPED actions here

		mpPACKML_STATE_STARTING:

			// Add STARTING actions here

			MpPackMLModule_Main.Command.StateComplete := TRUE;

		mpPACKML_STATE_IDLE:

			// Add IDLE actions here

		mpPACKML_STATE_SUSPENDING:

			// Add SUSPENDING actions here

			MpPackMLModule_Main.Command.StateComplete := TRUE;

		mpPACKML_STATE_SUSPENDED:

			// Add SUSPENDED actions here

		mpPACKML_STATE_UNSUSPENDING:

			// Add UNSUSPENDING actions here

			MpPackMLModule_Main.Command.StateComplete := TRUE;

		mpPACKML_STATE_EXECUTE:

			// Add EXECUTE actions here

		mpPACKML_STATE_STOPPING:

			// Add STOPPING actions here

			MpPackMLModule_Main.Command.StateComplete := TRUE;

		mpPACKML_STATE_ABORTING:

			// Add ABORTING actions here

			MpPackMLModule_Main.Command.StateComplete := TRUE;

		mpPACKML_STATE_ABORTED:

			// Add ABORTED actions here

		mpPACKML_STATE_HOLDING:

			// Add HOLDING actions here

			MpPackMLModule_Main.Command.StateComplete := TRUE;

		mpPACKML_STATE_HELD:

			// Add HELD actions here

		mpPACKML_STATE_UNHOLDING:

			// Add UNHOLDING actions here

			MpPackMLModule_Main.Command.StateComplete := TRUE;

		mpPACKML_STATE_COMPLETING:

			// Add COMPLETING actions here

			// NOTE: once COMPLETING actions that take more than one cyclic have been added, the below line
			// should be removed and replaced by the following line.
			MpPackMLModule_Main.Command.StateComplete := NOT MpPackMLModule_Main.Command.StateComplete;
			// MpPackMLModule_Main.Command.StateComplete := TRUE;

		mpPACKML_STATE_COMPLETE:

			// Add COMPLETE actions here

		mpPACKML_STATE_RESETTING:

			// Add RESETTING actions here

			MpPackMLModule_Main.Command.StateComplete := TRUE;

		mpPACKML_STATE_CLEARING:

			// Add CLEARING actions here

			MpPackMLModule_Main.Command.StateComplete := TRUE;

		mpPACKML_STATE_DEACTIVATING:

			// Add DEACTIVATING actions here

		mpPACKML_STATE_DEACTIVATED:

			// Add DEACTIVATED actions here

		mpPACKML_STATE_ACTIVATING:

			// Add ACTIVATING actions here

			MpPackMLModule_Main.Command.StateComplete := TRUE;

	END_CASE

END_ACTION
```

- Visualisation Logical/mappView (not shown)

### Package Logical/MachineControl - Package for Machine Control

### LICENSE.txt
```
MIT License

Copyright (c) 2022 B&R Industrial Automation

Permission is hereby granted, free of charge, to any person obtaining a copy
of this software and associated documentation files (the "Software"), to deal
in the Software without restriction, including without limitation the rights
to use, copy, modify, merge, publish, distribute, sublicense, and/or sell
copies of the Software, and to permit persons to whom the Software is
furnished to do so, subject to the following conditions:

The above copyright notice and this permission notice shall be included in all
copies or substantial portions of the Software.

THE SOFTWARE IS PROVIDED "AS IS", WITHOUT WARRANTY OF ANY KIND, EXPRESS OR
IMPLIED, INCLUDING BUT NOT LIMITED TO THE WARRANTIES OF MERCHANTABILITY,
FITNESS FOR A PARTICULAR PURPOSE AND NONINFRINGEMENT. IN NO EVENT SHALL THE
AUTHORS OR COPYRIGHT HOLDERS BE LIABLE FOR ANY CLAIM, DAMAGES OR OTHER
LIABILITY, WHETHER IN AN ACTION OF CONTRACT, TORT OR OTHERWISE, ARISING FROM,
OUT OF OR IN CONNECTION WITH THE SOFTWARE OR THE USE OR OTHER DEALINGS IN THE
SOFTWARE.
```

### AxisMgr.var - Local variables, used for all axes
```iecst
VAR
	i : {REDUND_UNREPLICABLE} USINT; (*Loop index variable*)
	ParameterState : {REDUND_UNREPLICABLE} ParameterStateEnum; (*Parameter handling state*)
	ConfigurationState : {REDUND_UNREPLICABLE} ConfigurationStateEnum; (*Configuration handling state*)
	State : {REDUND_UNREPLICABLE} StateEnum; (*OMAC based state machine*)
	AutomaticState : {REDUND_UNREPLICABLE} AutomaticStateEnum; (*Automatic handling state*)
	ManualState : {REDUND_UNREPLICABLE} ManualStateEnum; (*Manual handling state*)
	AxisControl : {REDUND_UNREPLICABLE} AxisControlType := (Status:=(StatusPointControl:=[0,1])); (*Single axis control type*)
	AxisSettings : {REDUND_UNREPLICABLE} AxisSettingsType; (*Single axis settings *)
END_VAR
(*Function Blocks*)
VAR
	MpRecipeRegParCfg : {REDUND_UNREPLICABLE} MpRecipeRegPar; (*Register function block for configuration values*)
	MpRecipeRegParPar : {REDUND_UNREPLICABLE} MpRecipeRegPar; (*Register function block for parameter values*)
	MpAlarmXCoreAxis : {REDUND_UNREPLICABLE} MpAlarmXCore; (*AlarmX Core function block*)
	MpAxisParameters : {REDUND_UNREPLICABLE} MpAxisBasicParType := (Distance:=70,Velocity:=100,Acceleration:=5000,Deceleration:=5000,Jog:=(Velocity:=70,Acceleration:=5000,Deceleration:=5000),AutoTune:=(MaxCurrentPercent:=50,MaxDistance:=720,MaxPositionError:=5)); (*Standard MpAxis parameter structure *)
	MpAxisBasicAppAxis : {REDUND_UNREPLICABLE} MpAxisBasic; (*MpAxis main function block*)
	ProcessConfigAX : {REDUND_UNREPLICABLE} MC_BR_ProcessConfig; (*Function block to read and write the axis configuration*)
	ProcessConfigACP : {REDUND_UNREPLICABLE} MC_BR_ProcessConfig; (*Function block to read and write the ACOPOS configuration*)
	IsHomedEdgePos : {REDUND_UNREPLICABLE} R_TRIG; (*Detecting rising edge for Homed*)
	InPositionEdgePos : {REDUND_UNREPLICABLE} R_TRIG; (*Detecting rising edge for InPosition*)
	ReferenceEdgePos : {REDUND_UNREPLICABLE} R_TRIG; (*Detecting rising edge for Referenced*)
	ZeroPendingAlarmsEdgePos : {REDUND_UNREPLICABLE} R_TRIG; (*Detecting rising edge when all alarms are cleared*)
	ProcessParamAX : {REDUND_UNREPLICABLE} MC_BR_ProcessParam; (*Function block to read and write the ACOPOS parameters*)
	AlarmSpeedNotSet : {REDUND_UNREPLICABLE} MpAlarmXAlarmControl; (*AlarmX control function block*)
END_VAR
(*Recipe*)
VAR
	ParametersEdit : {REDUND_UNREPLICABLE} AxisControlParametersType; (*Parameter structure used in recipe for edit*)
	ParametersPreview : {REDUND_UNREPLICABLE} AxisControlParametersType; (*Parameter structure used in recipe for preview*)
	MachineSettings : {REDUND_UNREPLICABLE} AxisMachineSettingsType; (*Machine settings structure*)
	MachineSettingsEdit : {REDUND_UNREPLICABLE} AxisMachineSettingsType; (*Machine settings structure used in recipe for edit*)
	MachineSettingsPreview : {REDUND_UNREPLICABLE} AxisMachineSettingsType; (*Machine settings structure used in recipe for preview*)
	AxisRecipe : {REDUND_UNREPLICABLE} AxisRecipeType; (*HMI interface structure*)
END_VAR
```

### AxisMgr.typ - Local data types
```iecst
(*Structure types*)

TYPE
	AxisSettingsType : 	STRUCT
		AxisFeatures : {REDUND_UNREPLICABLE} ARRAY[0..2]OF STRING[255]; (*Variable to write axis features into*)
		DriveConfiguration : {REDUND_UNREPLICABLE} McCfgPureVAxType; (*Drive configuration structure*)
		BaseConfiguration : {REDUND_UNREPLICABLE} McCfgAxType; (*Base axis type configuration *)
		BaseParam : {REDUND_UNREPLICABLE} McCfgAxMoveLimType; (*Base axis movement configuration*)
	END_STRUCT;
	AxisMachineSettingsType : {REDUND_UNREPLICABLE} 	STRUCT
		ReferencePosition : {REDUND_UNREPLICABLE} LREAL := 0; (*[mm] Axis position after reference*)
	END_STRUCT;
	AxisControlCommandType : {REDUND_UNREPLICABLE} 	STRUCT
		UpdatePreviewParameters : {REDUND_UNREPLICABLE} BOOL; (*Cmd to load new preview*)
		LoadRecipeParameters : {REDUND_UNREPLICABLE} BOOL; (*Load selected recipe file into active parameters *)
		SaveRecipeParameters : {REDUND_UNREPLICABLE} BOOL; (*Save current parameters*)
		Power : {REDUND_UNREPLICABLE} BOOL; (*Cmd power*)
		Reference : {REDUND_UNREPLICABLE} BOOL; (*Cmd home / reference*)
		MoveAbsolute : {REDUND_UNREPLICABLE} BOOL; (*Cmd move absolute*)
		MoveAdditive : {REDUND_UNREPLICABLE} BOOL; (*Cmd move additive*)
		MoveVelocity : {REDUND_UNREPLICABLE} BOOL; (*Cmd move velocity*)
		MoveToStart : {REDUND_UNREPLICABLE} BOOL; (*Cmd move the start position*)
		Abort : {REDUND_UNREPLICABLE} BOOL; (*Cmd abort*)
		Stop : {REDUND_UNREPLICABLE} BOOL; (*Cmd stop all movement*)
		Reset : {REDUND_UNREPLICABLE} BOOL; (*Cmd reset axis state*)
		JogPositive : {REDUND_UNREPLICABLE} BOOL; (*Cmd jog positive*)
		JogNegative : {REDUND_UNREPLICABLE} BOOL; (*Cmd jog negative*)
		Start : {REDUND_UNREPLICABLE} BOOL; (*Cmd start motion*)
		UpdateVelocity : {REDUND_UNREPLICABLE} BOOL; (*Cmd update velocity for automatic mode*)
	END_STRUCT;
	AxisControlParametersType : {REDUND_UNREPLICABLE} 	STRUCT
		HomePosition : {REDUND_UNREPLICABLE} LREAL := 0; (*[mm] Home Position*)
		Position : {REDUND_UNREPLICABLE} LREAL := 0; (*[mm] Position for absolute move*)
		Distance : {REDUND_UNREPLICABLE} LREAL := 50; (*[mm] Distance for relative move*)
		Velocity : {REDUND_UNREPLICABLE} REAL := 100; (*[mm/s] Velocity for absoluate and relative moves*)
		Acceleration : {REDUND_UNREPLICABLE} REAL := 360; (*[mm/s2] Acceleration for absoluate and relative moves*)
		Deceleration : {REDUND_UNREPLICABLE} REAL := 360; (*[mm/s2] Deceleration for absoluate and relative moves*)
		JogVelocity : {REDUND_UNREPLICABLE} REAL := 100; (*[mm/s] Velocity used when jogging the axis*)
		StopDeceleration : {REDUND_UNREPLICABLE} REAL := 720; (*[mm/s2] Deceleration for stopping*)
	END_STRUCT;
	AxisControlStatusType : {REDUND_UNREPLICABLE} 	STRUCT
		TaskName : {REDUND_UNREPLICABLE} STRING[80]; (*Current task name for configuration changes*)
		MachineSettingsName : {REDUND_UNREPLICABLE} STRING[255]; (*Category name for machine settings*)
		ProductSettingsName : {REDUND_UNREPLICABLE} STRING[255]; (*Category name for product settings*)
		Status : {REDUND_UNREPLICABLE} STRING[80]; (*Machine Status*)
		IsReady : {REDUND_UNREPLICABLE} BOOL; (*Axis is ready*)
		ErrorActive : {REDUND_UNREPLICABLE} BOOL; (*Error active*)
		Busy : {REDUND_UNREPLICABLE} BOOL; (*Cmd execution*)
		ReferenceRequired : {REDUND_UNREPLICABLE} BOOL; (*Reference cmd required*)
		Position : {REDUND_UNREPLICABLE} LREAL; (*Current position*)
		Velocity : {REDUND_UNREPLICABLE} REAL; (*Current position*)
		Current : {REDUND_UNREPLICABLE} REAL; (*Drive current*)
		LagError : {REDUND_UNREPLICABLE} LREAL; (*Axis lag error *)
		MotorTemperature : {REDUND_UNREPLICABLE} REAL; (*Motor temperature*)
		IsHomed : {REDUND_UNREPLICABLE} BOOL; (*Axis is referenced*)
		IsPowered : {REDUND_UNREPLICABLE} BOOL; (*Axis is powered*)
		PLCopenState : {REDUND_UNREPLICABLE} McAxisPLCopenStateEnum; (*Axis PLCopenState*)
		ModeManual : {REDUND_UNREPLICABLE} BOOL; (*Axis may be moved manually*)
		StatusPointControl : {REDUND_UNREPLICABLE} ARRAY[0..1]OF UINT; (*VC4 - Axis Manual/Auto control*)
	END_STRUCT;
	AxisControlType : {REDUND_UNREPLICABLE} 	STRUCT
		Command : {REDUND_UNREPLICABLE} AxisControlCommandType; (*Cmd structure*)
		Parameters : {REDUND_UNREPLICABLE} AxisControlParametersType; (*Parameter structure*)
		Status : {REDUND_UNREPLICABLE} AxisControlStatusType; (*Status structure*)
	END_STRUCT;
	AxisRecipeType : 	STRUCT
		EditDialogOpened : BOOL; (*HMI edit dialog open*)
		CreateDialogOpened : BOOL; (*HMI create dialog open*)
		SaveRecipe : BOOL; (*Cmd save current values*)
		LoadRecipe : BOOL; (*Cmd load exiting recipe*)
		CreateRecipe : BOOL; (*Cmd create new recipe*)
		State : AxisRecipeStepEnum; (*Recipe handling state*)
		CategoryDropdown : STRING[50]; (*HMI selector*)
	END_STRUCT;
END_TYPE

(*Enumerations*)

TYPE
	StateEnum :
		(
		STATE_INIT, (*Axis initialization state*)
		STATE_POWER_ON, (*Axis powering on state*)
		STATE_HOME, (*Axis homing state*)
		STATE_REFERENCE, (*Axis reference state*)
		STATE_MOVE_TO_HOME_POSITION, (*Axis moving to reference position state*)
		STATE_READY, (*Axis ready state*)
		STATE_MANUAL_OPERATION, (*Axis manual state*)
		STATE_AUTOMATIC_OPERATION, (*Axis automatic state*)
		STATE_STOPPING, (*Axis stopping state*)
		STATE_STOPPED, (*Axis stopped state*)
		STATE_ABORTING, (*Axis aborting state*)
		STATE_ABORTED, (*Axis aborted state*)
		STATE_CLEARING, (*Axis clearing state*)
		STATE_RESETTING (*Axis resetting state*)
		);
	ParameterStateEnum :
		(
		PAR_STATE_NOT_USED, (*Param initialization not used*)
		PAR_STATE_INIT, (*Param initialization state*)
		PAR_STATE_READ, (*Param read state*)
		PAR_STATE_WRITE, (*Param write state*)
		PAR_STATE_READY (*Param ready state*)
		);
	ConfigurationStateEnum :
		(
		CONFIG_STATE_NOT_USED, (*Config initialization not used*)
		CONFIG_STATE_INIT, (*Config initialization state*)
		CONFIG_STATE_READ, (*Config read state*)
		CONFIG_STATE_WRITE, (*Config write state*)
		CONFIG_STATE_READY (*Config ready state*)
		);
	ManualStateEnum :
		(
		MANUAL_STATE_IDLE, (*Idle state*)
		MANUAL_STATE_JOG, (*Jog state*)
		MANUAL_STATE_MOVE, (*Move state*)
		MANUAL_STATE_STOPPING (*Stopping state*)
		);
	AutomaticStateEnum :
		(
		AUTOMATIC_STATE_IDLE, (*Idle state*)
		AUTOMATIC_STATE_RUNNING (*Run state*)
		);
	AxisRecipeStepEnum :
		(
		REC_AXIS_WAIT, (*Wait state*)
		REC_AXIS_LOAD, (*Load product parameters*)
		REC_AXIS_SAVE, (*Save product parameters*)
		REC_AXIS_CREATE, (*Create new axis recipe*)
		REC_AXIS_STORE_MACH_SETTINGS, (*Save machine parameter settings*)
		REC_AXIS_FACTORY_RESET (*Factory reset*)
		);
END_TYPE
```

### AxisStateMachine.st - Generic state machine, used for all axes
```iecst
ACTION AxisStateMachine:

	InPositionEdgePos.CLK := MpAxisBasicAppAxis.InPosition;
	InPositionEdgePos();
	IsHomedEdgePos.CLK := MpAxisBasicAppAxis.IsHomed;
	IsHomedEdgePos();
	ReferenceEdgePos.CLK := AxisControl.Command.Reference;
	ReferenceEdgePos();
	ZeroPendingAlarmsEdgePos.CLK := (MpAlarmXCoreAxis.PendingAlarms = 0);
	ZeroPendingAlarmsEdgePos();

	CASE State OF
		STATE_STOPPING..STATE_RESETTING:
			// Nothing to do as we are already handling any stop or errors in these states

		ELSE
			IF ((MpAxisBasicAppAxis.Error) OR MpAlarmXCheckReaction(gMpLinkAlarmXCore, 'Error')) THEN
				// Check alarm reaction
				ResetAllAxisCommands;
				State := STATE_ABORTING;
			ELSIF ((NOT AxisControl.Command.Power) AND (State > STATE_POWER_ON)) THEN
				ResetAllAxisCommands;
				AxisControl.Status.Busy := TRUE;
				MpAxisBasicAppAxis.Power := FALSE;
				State := STATE_POWER_ON;
			END_IF

	END_CASE

	CASE State OF
		// Init state
		STATE_INIT:
			AxisControl.Status.Status := 'Initializing';
			ChangeConfiguration;
			ChangeParameter;
			IF (((ConfigurationState = CONFIG_STATE_READY) OR (ConfigurationState = CONFIG_STATE_NOT_USED)) AND ((ParameterState = PAR_STATE_READY) OR (ParameterState = PAR_STATE_NOT_USED)) AND (MpAxisBasicAppAxis.Active)) THEN
				AxisControl.Status.IsReady := TRUE;

				State := STATE_POWER_ON;
			END_IF

		// Power on the axis
		STATE_POWER_ON:
			AxisControl.Status.Status := 'Waiting for power on';
			IF (MpAxisBasicAppAxis.Info.ReadyToPowerOn) THEN
				MpAxisBasicAppAxis.Power := AxisControl.Command.Power;
			END_IF

			AxisControl.Status.Busy := MpAxisBasicAppAxis.Power;
			IF (MpAxisBasicAppAxis.PowerOn) THEN
				AxisControl.Status.Busy := FALSE;
				State := STATE_HOME;
			ELSE
				ChangeConfiguration;
			END_IF

		// Restore home position
		STATE_HOME:
			AxisControl.Status.Status := 'Waiting for home';
			IF ((NOT MpAxisBasicAppAxis.IsHomed) AND (MpAxisBasicAppAxis.PowerOn)) THEN
				AxisControl.Status.ReferenceRequired := TRUE;
				State := STATE_REFERENCE;
			END_IF

			IF (MpAxisBasicAppAxis.IsHomed) THEN
				AxisControl.Status.ReferenceRequired := FALSE;
				AxisControl.Status.Busy := FALSE;
				AxisControl.Command.Reference := FALSE;
				State := STATE_MOVE_TO_HOME_POSITION;
				ResetAllAxisCommands;
			END_IF

		// Create reference position
		STATE_REFERENCE:
			IF (AxisControl.Command.Reference) THEN
				AxisControl.Command.Reference := FALSE;
				MpAxisBasicAppAxis.Home := TRUE;
				AxisControl.Status.Busy := TRUE;
				MpAxisParameters.Homing.Mode := mcHOMING_DIRECT;
				MpAxisParameters.Homing.Position := MachineSettings.ReferencePosition;
			END_IF

			IF (IsHomedEdgePos.Q	= TRUE) THEN
				AxisControl.Status.ReferenceRequired := FALSE;
				State := STATE_MOVE_TO_HOME_POSITION;
				ResetAllAxisCommands;
			END_IF

		// Move to home position
		STATE_MOVE_TO_HOME_POSITION:
			AxisControl.Status.Status := 'Moving to home position';
			MpAxisParameters.Position := AxisControl.Parameters.HomePosition;
			MpAxisParameters.Direction := mcDIR_SHORTEST_WAY;
			MpAxisBasicAppAxis.MoveAbsolute := TRUE;
			IF (InPositionEdgePos.Q	= TRUE) THEN
				AxisControl.Status.Busy := FALSE;
				MpAxisBasicAppAxis.MoveAbsolute := FALSE;
				MpAxisParameters.Direction := mcDIR_POSITIVE;
				State := STATE_READY;
			END_IF

		// In this State the module is error free and ready for a command (manual or automatic)
		STATE_READY:
			AxisControl.Status.Status := 'Ready';
			AxisControl.Status.Busy := FALSE;
			IF (ReferenceEdgePos.Q) THEN
				State := STATE_REFERENCE;
			ELSIF ((NOT MpAlarmXCheckReaction(gMpLinkAlarmXCore, 'Warning')) AND (AutomaticCommand(AxisControl.Command))) THEN
				State := STATE_AUTOMATIC_OPERATION;
			ELSIF (ManualCommand(AxisControl.Command)) THEN
				State := STATE_MANUAL_OPERATION;
			END_IF

		// Axis can be moved manually / jogged
		STATE_MANUAL_OPERATION:
			AxisControl.Status.Status := 'Manual running';
			AxisControl.Status.Busy := TRUE;
			AxisManual;

		// Axis put into automatic mode / camming
		STATE_AUTOMATIC_OPERATION:
			AxisControl.Status.Status := 'Automatic running';
			AxisControl.Status.Busy := TRUE;
			IF MpAlarmXCheckReaction(gMpLinkAlarmXCore, 'Error') THEN
				AxisControl.Command.Stop := TRUE;
			END_IF

			AxisAutomatic;

		// In this State the module will attempt to bring the axis to a controlled stop.
		STATE_STOPPING:
			AxisControl.Status.Status := 'Stopping';

			// Stop the axis if it is powered on
			MpAxisBasicAppAxis.Stop := MpAxisBasicAppAxis.PowerOn;
			MpAxisParameters.Stop.Deceleration := AxisControl.Parameters.StopDeceleration;
			IF ((NOT MpAxisBasicAppAxis.PowerOn) OR (MpAxisBasicAppAxis.Stopped)) THEN
				MpAxisBasicAppAxis.Stop := FALSE;
				State := STATE_STOPPED;
			END_IF

		// In this State the module is powered on and at standstill.
		STATE_STOPPED:
			State := STATE_RESETTING;

		// In this State the module will bring the axis to a rapid stop
		STATE_ABORTING:
			MpAxisParameters.Stop.Deceleration := 0;
			MpAxisBasicAppAxis.Stop := MpAxisBasicAppAxis.PowerOn;
			IF ((NOT MpAxisBasicAppAxis.PowerOn) OR (MpAxisBasicAppAxis.Stopped)) THEN
				MpAxisBasicAppAxis.Stop := FALSE;
				IF (MpAlarmXCheckReaction(gMpLinkAlarmXCore, 'SafetyError')) THEN
					// Safety errors also power off the axis
					MpAxisBasicAppAxis.Power := FALSE;
					IF (NOT MpAxisBasicAppAxis.PowerOn) THEN
						State := STATE_ABORTED;
					END_IF
				ELSE
					State := STATE_ABORTED;
				END_IF
			END_IF

		STATE_ABORTED:
			State := STATE_CLEARING;

		STATE_CLEARING:
			State := STATE_RESETTING;

		// In this State the module attempts to clear any outstanding errors.  No hazardous motion should occur in this State.
		STATE_RESETTING:
			ResetAllAxisCommands;
			IF (AxisControl.Command.Reset) OR ((NOT MpAlarmXCheckReaction(gMpLinkAlarmXCore, 'Error')) AND ZeroPendingAlarmsEdgePos.Q) THEN
				AxisControl.Status.Busy := TRUE;
				AxisControl.Command.Reset := FALSE;
				MpAxisBasicAppAxis.ErrorReset := TRUE;
				AxisReset;
				ManualState := MANUAL_STATE_IDLE;
				AutomaticState := AUTOMATIC_STATE_IDLE;
			ELSE
				MpAxisBasicAppAxis.ErrorReset := FALSE;
			END_IF

			IF ((NOT MpAxisBasicAppAxis.Error) AND (NOT MpAlarmXCheckReaction(gMpLinkAlarmXCore, 'Error'))) THEN
				AxisControl.Status.Busy := FALSE;
				IF (NOT MpAxisBasicAppAxis.PowerOn) THEN
					State := STATE_POWER_ON;
				ELSIF (MpAxisBasicAppAxis.IsHomed) THEN
					State := STATE_READY;
				ELSE
					State := STATE_HOME;
				END_IF
			END_IF

	END_CASE

	// Cyclic function block calls
	MpAxisBasicAppAxis.Parameters := ADR(MpAxisParameters);
	MpAxisBasicAppAxis();

	// Status assignments
	AxisControl.Status.ErrorActive := MpAxisBasicAppAxis.Error OR (MpAlarmXCheckReaction(gMpLinkAlarmXCore, 'Error'));
	AxisControl.Status.IsHomed := MpAxisBasicAppAxis.IsHomed;
	AxisControl.Status.IsPowered := MpAxisBasicAppAxis.PowerOn;
	AxisControl.Status.PLCopenState := MpAxisBasicAppAxis.Info.PLCopenState;
	AxisControl.Status.Position := MpAxisBasicAppAxis.Position;
	AxisControl.Status.Velocity := MpAxisBasicAppAxis.Velocity;
	AxisControl.Status.ModeManual := (State <> STATE_AUTOMATIC_OPERATION);
	//VC4 related code
	AxisControl.Status.StatusPointControl[0].0 := NOT AxisControl.Status.StatusPointControl[1].0;
	AxisControl.Status.StatusPointControl[0].1 := NOT AxisControl.Status.ModeManual;

END_ACTION

ACTION ResetAllAxisCommands:

	MpAxisBasicAppAxis.MoveAbsolute := FALSE;
	MpAxisBasicAppAxis.MoveAdditive := FALSE;
	MpAxisBasicAppAxis.MoveVelocity := FALSE;
	MpAxisBasicAppAxis.ReleaseBrake := FALSE;
	MpAxisBasicAppAxis.ErrorReset := FALSE;
	MpAxisBasicAppAxis.JogPositive := FALSE;
	MpAxisBasicAppAxis.JogNegative := FALSE;
	MpAxisBasicAppAxis.Home := FALSE;

END_ACTION
```

### Recipe.st - Recipe handling
```iecst
ACTION RecipeInit:

	// Register the variables with the recipe system
	AxisControl.Status.ProductSettingsName := AxisControl.Status.TaskName;
	brsstrcat(ADR(AxisControl.Status.ProductSettingsName), ADR(':ParametersPreview'));
	MpRecipeRegParPar.MpLink := ADR(gMpLinkRecipeXml);
	MpRecipeRegParPar.Enable := TRUE;
	MpRecipeRegParPar.PVName := ADR(AxisControl.Status.ProductSettingsName);
	MpRecipeRegParPar.Category := ADR(PARAMETERS_CATEGORY);
	MpRecipeRegParPar();
	ParametersPreview;
	ParametersEdit;

	AxisControl.Status.MachineSettingsName := AxisControl.Status.TaskName;
	brsstrcat(ADR(AxisControl.Status.MachineSettingsName), ADR(':MachineSettingsPreview'));
	MpRecipeRegParCfg.MpLink := ADR(gMpLinkRecipeXml);
	MpRecipeRegParCfg.Enable := TRUE;
	MpRecipeRegParCfg.PVName := ADR(AxisControl.Status.MachineSettingsName);
	MpRecipeRegParCfg.Category := ADR(MACHINE_CONFIGURATION_CATEGORY);
	MpRecipeRegParCfg();
	MachineSettingsPreview;
	MachineSettingsEdit;

	// Activate RegPar FUBs
	WHILE NOT(MpRecipeRegParPar.Active OR MpRecipeRegParPar.Error) DO
		MpRecipeRegParPar();
	END_WHILE
	WHILE NOT(MpRecipeRegParCfg.Active OR MpRecipeRegParCfg.Error) DO
		MpRecipeRegParCfg();
	END_WHILE

END_ACTION

ACTION RecipeCyclic:

	// HMI support handling
	IF (AxisRecipe.EditDialogOpened OR AxisRecipe.CreateDialogOpened) THEN
		IF (brsstrcmp(ADR(AxisRecipe.CategoryDropdown), ADR('Product')) = 0) THEN
			ParametersEdit := ParametersPreview;
		ELSIF (brsstrcmp(ADR(AxisRecipe.CategoryDropdown), ADR('Machine')) = 0) THEN
			MachineSettingsEdit := MachineSettingsPreview;
		END_IF
		AxisRecipe.EditDialogOpened := FALSE;
		AxisRecipe.CreateDialogOpened := FALSE;
	END_IF

	CASE AxisRecipe.State OF
		// Wait state
		REC_AXIS_WAIT:
			IF AxisRecipe.CreateRecipe THEN
				AxisRecipe.State := REC_AXIS_CREATE;
				AxisRecipe.CreateRecipe := FALSE;
			ELSIF AxisRecipe.SaveRecipe THEN
				AxisRecipe.State := REC_AXIS_SAVE;
				AxisRecipe.SaveRecipe := FALSE;
			ELSIF AxisRecipe.LoadRecipe THEN
				AxisRecipe.State := REC_AXIS_LOAD;
				AxisRecipe.LoadRecipe := FALSE;
			END_IF
		// Create recipe state
		REC_AXIS_CREATE:
			IF (brsstrcmp(ADR(AxisRecipe.CategoryDropdown), ADR('Product')) = 0) THEN
				ParametersPreview := ParametersEdit;
			ELSIF (brsstrcmp(ADR(AxisRecipe.CategoryDropdown), ADR('Machine')) = 0) THEN
				MachineSettingsPreview := MachineSettingsEdit;
			END_IF
			AxisRecipe.State := REC_AXIS_WAIT;
		// Load recipe state
		REC_AXIS_LOAD:
			IF (brsstrcmp(ADR(AxisRecipe.CategoryDropdown), ADR('Product')) = 0) THEN
				AxisControl.Parameters := ParametersPreview;
			ELSIF (brsstrcmp(ADR(AxisRecipe.CategoryDropdown), ADR('Machine')) = 0) THEN
				MachineSettings := MachineSettingsPreview;
			END_IF
			AxisRecipe.State := REC_AXIS_WAIT;
		// Save recipe state
		REC_AXIS_SAVE:
			IF (brsstrcmp(ADR(AxisRecipe.CategoryDropdown), ADR('Product')) = 0) THEN
				ParametersPreview := ParametersEdit;
			ELSIF (brsstrcmp(ADR(AxisRecipe.CategoryDropdown), ADR('Machine')) = 0) THEN
				MachineSettingsPreview := MachineSettingsEdit;
			END_IF
			AxisRecipe.State := REC_AXIS_WAIT;

	END_CASE;

	// Cyclic function block calls
	MpRecipeRegParPar.MpLink := ADR(gMpLinkRecipeXml);
	IF (AxisControl.Status.ProductSettingsName = '') THEN
		AxisControl.Status.ProductSettingsName := AxisControl.Status.TaskName;
		brsstrcat(ADR(AxisControl.Status.ProductSettingsName), ADR(':ParametersPreview'));
	END_IF
	MpRecipeRegParPar.PVName := ADR(AxisControl.Status.ProductSettingsName);
	MpRecipeRegParPar.Category := ADR(PARAMETERS_CATEGORY);
	MpRecipeRegParPar();

	MpRecipeRegParCfg.MpLink := ADR(gMpLinkRecipeXml);
	IF (AxisControl.Status.MachineSettingsName = '') THEN
		AxisControl.Status.MachineSettingsName := AxisControl.Status.TaskName;
		brsstrcat(ADR(AxisControl.Status.MachineSettingsName), ADR(':MachineSettingsPreview'));
	END_IF

	MpRecipeRegParCfg.PVName := ADR(AxisControl.Status.MachineSettingsName);
	MpRecipeRegParCfg.Category := ADR(MACHINE_CONFIGURATION_CATEGORY);
	MpRecipeRegParCfg();

END_ACTION
```

### ChangeConfiguration.st - Changes the axis configuration at runtime
```iecst
ACTION ConfigurationInit:
	// Initalize drive configuration
	AxisSettings.DriveConfiguration.PureVirtualAxis.AxisFeatures.FeatureReference.DataAddress := ADR(AxisSettings.AxisFeatures);
	AxisSettings.DriveConfiguration.PureVirtualAxis.AxisFeatures.FeatureReference.NumberOfArrayElements := SIZEOF(AxisSettings.AxisFeatures)/SIZEOF(AxisSettings.AxisFeatures[0]);
	AxisSettings.DriveConfiguration.PureVirtualAxis.AxisFeatures.FeatureReference.NumberOfElements := 0;
	i := 0;
	WHILE ((i <= SIZEOF(AxisSettings.AxisFeatures)/SIZEOF(AxisSettings.AxisFeatures[0])) AND (AxisSettings.AxisFeatures[i] <> '')) DO
		i := i + 1;
	END_WHILE
	AxisSettings.DriveConfiguration.PureVirtualAxis.AxisFeatures.FeatureReference.NumberOfElements := i;

	ProcessConfigAX.DataAddress := ADR(AxisSettings.BaseConfiguration);
	ProcessConfigAX.DataType := mcCFG_AX;

	ProcessConfigACP.DataAddress := ADR(AxisSettings.DriveConfiguration);
	ProcessConfigACP.DataType := mcCFG_PURE_V_AX;

	ConfigurationState := CONFIG_STATE_INIT;

END_ACTION

ACTION ChangeConfiguration:

	CASE ConfigurationState OF
		CONFIG_STATE_INIT:

			// Assign string for the name
			ProcessConfigACP.Name := MpAxisBasicAppAxis.Info.HardwareInfo.Axis.ConfigElementLocation;
			ProcessConfigAX.Name := MpAxisBasicAppAxis.Info.HardwareInfo.Axis.AxisName;

			IF (MpAxisBasicAppAxis.Active) THEN
				ConfigurationState := CONFIG_STATE_READ;
			END_IF

		CONFIG_STATE_READ:
			// Read the current configuration
			ProcessConfigACP.Mode := mcPCM_LOAD;
			ProcessConfigACP.Execute := TRUE;

			ProcessConfigAX.Mode := mcPCM_LOAD;
			ProcessConfigAX.Execute := TRUE;
			IF (ProcessConfigACP.Done) AND (ProcessConfigAX.Done) THEN
				ProcessConfigACP.Execute := FALSE;
				ProcessConfigAX.Execute := FALSE;
				ConfigurationState := CONFIG_STATE_READY;
			END_IF

		CONFIG_STATE_WRITE:
			// Write the configuration after changes
			ProcessConfigACP.Mode := mcPCM_SAVE;
			ProcessConfigACP.Execute := TRUE;

			ProcessConfigAX.Mode := mcPCM_SAVE;
			ProcessConfigAX.Execute := TRUE;
			IF (ProcessConfigACP.Done) AND (ProcessConfigAX.Done) THEN
				ProcessConfigACP.Execute := FALSE;
				ProcessConfigAX.Execute := FALSE;
				ConfigurationState := CONFIG_STATE_READY;
			END_IF

		CONFIG_STATE_READY:

	END_CASE

	// Cyclic function block calls
	AxisSettings.DriveConfiguration.PureVirtualAxis.AxisFeatures.FeatureReference.DataAddress := ADR(AxisSettings.AxisFeatures);
	ProcessConfigAX.DataAddress := ADR(AxisSettings.BaseConfiguration);
	ProcessConfigACP.DataAddress := ADR(AxisSettings.DriveConfiguration);
	ProcessConfigACP();
	ProcessConfigAX();

END_ACTION

ACTION ParameterInit:
	// Initalize drive parameter
	ProcessParamAX.DataAddress := ADR(AxisSettings.BaseParam);
	ProcessParamAX.DataType := mcCFG_AX_MOVE_LIM;

	ParameterState := PAR_STATE_INIT;

END_ACTION

ACTION ChangeParameter:

	CASE ParameterState OF
		PAR_STATE_INIT:
			// Wait state
			ProcessParamAX.Component := MpAxisBasicAppAxis.MpLink;

			IF (MpAxisBasicAppAxis.Active) THEN
				ParameterState := PAR_STATE_READ;
			END_IF

		PAR_STATE_READ:
			// Read current parameter values
			ProcessParamAX.Mode := mcPPM_READ;
			ProcessParamAX.Execute := TRUE;

			IF (ProcessParamAX.Done) THEN
				ProcessParamAX.Execute := FALSE;
				ParameterState := PAR_STATE_READY;
			END_IF

		PAR_STATE_WRITE:
			// Write new parameter values
			ProcessParamAX.Mode := mcPPM_WRITE;
			ProcessParamAX.Execute := TRUE;

			IF (ProcessParamAX.Done) THEN
				ProcessParamAX.Execute := FALSE;
				ParameterState := PAR_STATE_READY;
			END_IF

		PAR_STATE_READY:

	END_CASE

	ProcessParamAX.DataAddress := ADR(AxisSettings.BaseParam);
	ProcessParamAX();

END_ACTION
```

### Package Logical/MachineControl/AxisTemplate - Package for mapp Axis Framework Template

### Program Logical/MachineControl/AxisTemplate/AxisMgr (IEC) - Axis control

#### AxisMgr.st - Init, cyclic, exit code
```iecst
//***********************************************************************
// Copyright: B&R Industrial Automation GmbH
// Author: B&R Industrial Automation GmbH
// Created: April 12, 2022
// Description: Tasks for axis control.
//***********************************************************************

PROGRAM _INIT

	// Read current task name for category setup
	ST_name(0, ADR(AxisControl.Status.TaskName), 0);

	// Call initialization actions
	RecipeInit;
	ConfigurationInit;
	ParameterInit;
	AxisInit;

	// Call initialization variables
	RestorePosition_AxisTemplate;

	// Initialize homing mode
	MpAxisParameters.Homing.Mode := mcHOMING_DEFAULT;

	// Enable mapp function blocks
	MpAxisBasicAppAxis.Enable := TRUE;
	MpAlarmXCore_0.Enable := TRUE;

END_PROGRAM

PROGRAM _CYCLIC

	MpAxisBasicAppAxis.MpLink := ADR(gAxisTemplate);

	// Call all actions
	SimulationControl;
	AxisStateMachine;
	AxisCyclic;
	RecipeCyclic;

	// Assign MpLink
	MpAlarmXCore_0.MpLink := ADR(gAlarmXCore_AxisTemplate);

	// Call function block
	MpAlarmXCore_0();

END_PROGRAM

PROGRAM _EXIT

	// Disable the function blocls to unlink the MpLinks.
	// Do NOT disable MpAxisBasic, as this can cause problems during project transfer.
	MpRecipeRegPar_Par.Enable := FALSE;
	MpRecipeRegPar_Cfg.Enable := FALSE;
	MpAlarmXCore_0.Enable := FALSE;

	// Call function blocks
	MpRecipeRegPar_Par();
	MpRecipeRegPar_Cfg();
	MpAlarmXCore_0();

END_PROGRAM
```

#### Variables.var - Local variables, specific to this axis
```iecst
VAR RETAIN
	RestorePosition_AxisTemplate : {REDUND_UNREPLICABLE} McAcpAxRestorePosType; (*Data structure for retsore position mode*)
END_VAR
```

#### AxisControlModes.st - Code that is specific to this axis
```iecst
ACTION AxisInit:
	// Action call during init
END_ACTION

ACTION AxisCyclic:
	// Cyclic action call
END_ACTION

ACTION AxisManual:
	// Action handling manual axis control
	MpAxisParameters.Jog.Velocity := AxisControl.Parameters.JogVelocity;
	MpAxisParameters.Velocity := AxisControl.Parameters.Velocity;
	MpAxisParameters.Position := AxisControl.Parameters.Position;
	MpAxisParameters.Distance := AxisControl.Parameters.Distance;
	MpAxisParameters.Acceleration := AxisControl.Parameters.Acceleration;
	MpAxisParameters.Deceleration := AxisControl.Parameters.Deceleration;
	MpAxisParameters.Stop.Deceleration := AxisControl.Parameters.StopDeceleration;

	CASE ManualState OF
		// Wait state
		MANUAL_STATE_IDLE:
			IF ((AxisControl.Command.JogNegative) OR (AxisControl.Command.JogPositive)) THEN
				ManualState := MANUAL_STATE_JOG;
			ELSIF ((AxisControl.Command.MoveAbsolute) OR (AxisControl.Command.MoveAdditive) OR (AxisControl.Command.MoveVelocity)) THEN
				MpAxisBasicAppAxis.MoveAbsolute := AxisControl.Command.MoveAbsolute;
				MpAxisBasicAppAxis.MoveAdditive := AxisControl.Command.MoveAdditive;
				MpAxisBasicAppAxis.MoveVelocity := AxisControl.Command.MoveVelocity;
				AxisControl.Command.MoveAbsolute := FALSE;
				AxisControl.Command.MoveAdditive := FALSE;
				ManualState := MANUAL_STATE_MOVE;
			ELSE
				State := STATE_READY;
			END_IF
			// Jog state
		MANUAL_STATE_JOG:
			MpAxisBasicAppAxis.JogNegative := AxisControl.Command.JogNegative;
			MpAxisBasicAppAxis.JogPositive := AxisControl.Command.JogPositive;
			IF (AxisControl.Command.Stop) THEN
				AxisControl.Command.Stop := FALSE;
				MpAxisBasicAppAxis.Stop := TRUE;
				ManualState := MANUAL_STATE_STOPPING;
			ELSIF ((NOT AxisControl.Command.JogNegative) AND (NOT AxisControl.Command.JogPositive)) THEN
				MpAxisBasicAppAxis.Stop := FALSE;
				MpAxisBasicAppAxis.JogPositive := FALSE;
				MpAxisBasicAppAxis.JogNegative := FALSE;
				ManualState := MANUAL_STATE_STOPPING;
			END_IF
			// Direct move state
		MANUAL_STATE_MOVE:
			IF (AxisControl.Command.Stop) THEN
				MpAxisBasicAppAxis.MoveAbsolute := FALSE;
				MpAxisBasicAppAxis.MoveAdditive := FALSE;
				AxisControl.Command.Stop := FALSE;
				MpAxisBasicAppAxis.Stop := TRUE;
				ManualState := MANUAL_STATE_STOPPING;
			ELSIF (InPositionEdgePos.Q) THEN
				MpAxisBasicAppAxis.MoveAbsolute := FALSE;
				MpAxisBasicAppAxis.MoveAdditive := FALSE;
				ManualState := MANUAL_STATE_IDLE;
				State := STATE_READY;
			ELSIF (((NOT AxisControl.Command.MoveVelocity) AND (NOT MpAxisBasicAppAxis.MoveAbsolute) AND (NOT MpAxisBasicAppAxis.MoveAdditive)) OR AxisControl.Status.ErrorActive)	THEN
				MpAxisBasicAppAxis.MoveVelocity := FALSE;
				ManualState := MANUAL_STATE_STOPPING;
			ELSIF ((AxisControl.Command.JogNegative) OR (AxisControl.Command.JogPositive)) THEN
				MpAxisBasicAppAxis.MoveAbsolute := FALSE;
				MpAxisBasicAppAxis.MoveAdditive := FALSE;
				ManualState := MANUAL_STATE_JOG;
			END_IF
			// Stopping active movements
		MANUAL_STATE_STOPPING:
			MpAxisBasicAppAxis.JogNegative := FALSE;
			MpAxisBasicAppAxis.JogPositive := FALSE;
			MpAxisBasicAppAxis.MoveAbsolute := FALSE;
			MpAxisBasicAppAxis.MoveAdditive := FALSE;
			AxisControl.Command.MoveVelocity := FALSE;
			MpAxisBasicAppAxis.Stop := TRUE;

			IF (NOT MpAxisBasicAppAxis.MoveActive) THEN
				MpAxisBasicAppAxis.Stop := FALSE;
				MpAxisBasicAppAxis.MoveVelocity := FALSE;
				ManualState := MANUAL_STATE_IDLE;
				State := STATE_READY;
			END_IF
	END_CASE

END_ACTION

ACTION AxisAutomatic:

	CASE AutomaticState OF
		AUTOMATIC_STATE_IDLE:
			IF (AxisControl.Command.Start) THEN
				AutomaticState := AUTOMATIC_STATE_RUNNING;
			END_IF

		AUTOMATIC_STATE_RUNNING:
			MpAxisBasicAppAxis.MoveVelocity := TRUE;
			MpAxisParameters.Acceleration := AxisControl.Parameters.Acceleration;
			MpAxisParameters.Deceleration := AxisControl.Parameters.Deceleration;
			MpAxisParameters.Velocity := ABS(AxisControl.Parameters.Velocity);
			IF (AxisControl.Parameters.Velocity < 0) THEN
				MpAxisParameters.Direction := mcDIR_NEGATIVE;
			ELSE
				MpAxisParameters.Direction := mcDIR_POSITIVE;
			END_IF

			IF ((NOT AxisControl.Command.Start) OR (AxisControl.Command.Stop)) THEN
				AxisControl.Command.Start := FALSE;
				AxisControl.Command.Stop := FALSE;
				MpAxisBasicAppAxis.MoveVelocity := FALSE;
				State := STATE_READY;
				AutomaticState := AUTOMATIC_STATE_IDLE;
			ELSIF (AxisControl.Command.UpdateVelocity) THEN
				AxisControl.Command.UpdateVelocity := FALSE;
				MpAxisBasicAppAxis.Update := TRUE;
			ELSIF (MpAxisBasicAppAxis.UpdateDone) THEN
				MpAxisBasicAppAxis.Update := FALSE;
			END_IF
	END_CASE

END_ACTION

ACTION AxisReset:
	// AxisReset action call
END_ACTION
```

#### SimulationControl.st - Simulation handling
```iecst
ACTION SimulationControl:

	// Automatic settings when project is in simulation
	IF NOT (DiagCpuIsARsim() OR DiagCpuIsSimulated()) THEN
		RETURN;
	END_IF

	IF ((MpAxisBasic_0.IsHomed = FALSE) AND (MpAxisBasic_0.Home = FALSE)) THEN
		AxisControl.Command.Reference := TRUE;
	END_IF

END_ACTION
```

#### ManualCommand.st - Defines conditions for manual mode
```iecst
// Returns True if a manual command is active, false otherwise
FUNCTION ManualCommand

	ManualCommand := Commands.JogNegative OR Commands.JogPositive OR Commands.MoveAbsolute OR Commands.MoveAdditive OR Commands.MoveVelocity;

END_FUNCTION
```

#### AutomaticCommand.st - Defines conditions for automatic mode
```iecst
// Returns True if an automatic command is active
FUNCTION AutomaticCommand

	AutomaticCommand := Commands.Start;

END_FUNCTION
```

- AxisMgr.var (reference to Logical/MachineControl/AxisReferencedFiles/AxisMgr.var)

- AxisMgr.typ (reference to Logical/MachineControl/AxisReferencedFiles/AxisMgr.typ)

- AxisStateMachine.st (reference to Logical/MachineControl/AxisReferencedFiles/AxisStateMachine.st)

- ChangeConfiguration.st (reference to Logical/MachineControl/AxisReferencedFiles/ChangeConfiguration.st)

- Recipe.st (reference to Logical/MachineControl/AxisReferencedFiles/Recipe.st)

#### AxisMgr.typ - not listed in the package file held
```iecst
(*Structure types*)

TYPE
	AxisSettingsType : 	STRUCT
		AxisFeatures : {REDUND_UNREPLICABLE} ARRAY[0..2]OF STRING[255]; (*Variable to write axis features into*)
		DriveConfiguration : {REDUND_UNREPLICABLE} McCfgPureVAxType; (*Drive configuration structure*)
		BaseConfiguration : {REDUND_UNREPLICABLE} McCfgAxType; (*Base axis type configuration *)
		BaseParam : {REDUND_UNREPLICABLE} McCfgAxMoveLimType; (*Base axis movement configuration*)
	END_STRUCT;
	AxisMachineSettingsType : {REDUND_UNREPLICABLE} 	STRUCT
		ReferencePosition : {REDUND_UNREPLICABLE} LREAL := 0; (*[mm] Axis position after reference*)
	END_STRUCT;
	AxisControlCommandType : {REDUND_UNREPLICABLE} 	STRUCT
		UpdatePreviewParameters : {REDUND_UNREPLICABLE} BOOL; (*Cmd to load new preview*)
		LoadRecipeParameters : {REDUND_UNREPLICABLE} BOOL; (*Load selected recipe file into active parameters *)
		SaveRecipeParameters : {REDUND_UNREPLICABLE} BOOL; (*Save current parameters*)
		Power : {REDUND_UNREPLICABLE} BOOL; (*Cmd power*)
		Reference : {REDUND_UNREPLICABLE} BOOL; (*Cmd home / reference*)
		MoveAbsolute : {REDUND_UNREPLICABLE} BOOL; (*Cmd move absolute*)
		MoveAdditive : {REDUND_UNREPLICABLE} BOOL; (*Cmd move additive*)
		MoveVelocity : {REDUND_UNREPLICABLE} BOOL; (*Cmd move velocity*)
		MoveToStart : {REDUND_UNREPLICABLE} BOOL; (*Cmd move the start position*)
		Abort : {REDUND_UNREPLICABLE} BOOL; (*Cmd abort*)
		Stop : {REDUND_UNREPLICABLE} BOOL; (*Cmd stop all movement*)
		Reset : {REDUND_UNREPLICABLE} BOOL; (*Cmd reset axis state*)
		JogPositive : {REDUND_UNREPLICABLE} BOOL; (*Cmd jog positive*)
		JogNegative : {REDUND_UNREPLICABLE} BOOL; (*Cmd jog negative*)
		Start : {REDUND_UNREPLICABLE} BOOL; (*Cmd start motion*)
		UpdateVelocity : {REDUND_UNREPLICABLE} BOOL; (*Cmd update velocity for automatic mode*)
	END_STRUCT;
	AxisControlParametersType : {REDUND_UNREPLICABLE} 	STRUCT
		HomePosition : {REDUND_UNREPLICABLE} LREAL := 0; (*[mm] Home Position*)
		Position : {REDUND_UNREPLICABLE} LREAL := 0; (*[mm] Position for absolute move*)
		Distance : {REDUND_UNREPLICABLE} LREAL := 50; (*[mm] Distance for relative move*)
		Velocity : {REDUND_UNREPLICABLE} REAL := 100; (*[mm/s] Velocity for absoluate and relative moves*)
		Acceleration : {REDUND_UNREPLICABLE} REAL := 360; (*[mm/s2] Acceleration for absoluate and relative moves*)
		Deceleration : {REDUND_UNREPLICABLE} REAL := 360; (*[mm/s2] Deceleration for absoluate and relative moves*)
		JogVelocity : {REDUND_UNREPLICABLE} REAL := 100; (*[mm/s] Velocity used when jogging the axis*)
		StopDeceleration : {REDUND_UNREPLICABLE} REAL := 720; (*[mm/s2] Deceleration for stopping*)
	END_STRUCT;
	AxisControlStatusType : {REDUND_UNREPLICABLE} 	STRUCT
		TaskName : {REDUND_UNREPLICABLE} STRING[80]; (*Current task name for configuration changes*)
		MachineSettingsName : {REDUND_UNREPLICABLE} STRING[255]; (*Category name for machine settings*)
		ProductSettingsName : {REDUND_UNREPLICABLE} STRING[255]; (*Category name for product settings*)
		Status : {REDUND_UNREPLICABLE} STRING[80]; (*Machine Status*)
		IsReady : {REDUND_UNREPLICABLE} BOOL; (*Axis is ready*)
		ErrorActive : {REDUND_UNREPLICABLE} BOOL; (*Error active*)
		Busy : {REDUND_UNREPLICABLE} BOOL; (*Cmd execution*)
		ReferenceRequired : {REDUND_UNREPLICABLE} BOOL; (*Reference cmd required*)
		Position : {REDUND_UNREPLICABLE} LREAL; (*Current position*)
		Velocity : {REDUND_UNREPLICABLE} REAL; (*Current position*)
		Current : {REDUND_UNREPLICABLE} REAL; (*Drive current*)
		LagError : {REDUND_UNREPLICABLE} LREAL; (*Axis lag error *)
		MotorTemperature : {REDUND_UNREPLICABLE} REAL; (*Motor temperature*)
		IsHomed : {REDUND_UNREPLICABLE} BOOL; (*Axis is referenced*)
		IsPowered : {REDUND_UNREPLICABLE} BOOL; (*Axis is powered*)
		PLCopenState : {REDUND_UNREPLICABLE} McAxisPLCopenStateEnum; (*Axis PLCopenState*)
		ModeManual : BOOL; (*Axis may be moved manually*)
		StatusPointControl : ARRAY[0..1]OF UINT; (*VC4 - Axis Manual/Auto control*)
	END_STRUCT;
	AxisControlType : {REDUND_UNREPLICABLE} 	STRUCT
		Command : {REDUND_UNREPLICABLE} AxisControlCommandType; (*Cmd structure*)
		Parameters : {REDUND_UNREPLICABLE} AxisControlParametersType; (*Parameter structure*)
		Status : {REDUND_UNREPLICABLE} AxisControlStatusType; (*Status structure*)
	END_STRUCT;
	AxisRecipeType : 	STRUCT
		EditDialogOpened : BOOL; (*HMI edit dialog open*)
		CreateDialogOpened : BOOL; (*HMI create dialog open*)
		SaveRecipe : BOOL; (*Cmd save current values*)
		LoadRecipe : BOOL; (*Cmd load exiting recipe*)
		CreateRecipe : BOOL; (*Cmd create new recipe*)
		State : AxisRecipeStepEnum; (*Recipe handling state*)
		CategoryDropdown : STRING[50]; (*HMI selector*)
	END_STRUCT;
END_TYPE

(*Enumerations*)

TYPE
	StateEnum :
		(
		STATE_INIT, (*Axis initialization state*)
		STATE_POWER_ON, (*Axis powering on state*)
		STATE_HOME, (*Axis homing state*)
		STATE_REFERENCE, (*Axis reference state*)
		STATE_MOVE_TO_HOME_POSITION, (*Axis moving to reference position state*)
		STATE_READY, (*Axis ready state*)
		STATE_MANUAL_OPERATION, (*Axis manual state*)
		STATE_AUTOMATIC_OPERATION, (*Axis automatic state*)
		STATE_STOPPING, (*Axis stopping state*)
		STATE_STOPPED, (*Axis stopped state*)
		STATE_ABORTING, (*Axis aborting state*)
		STATE_ABORTED, (*Axis aborted state*)
		STATE_CLEARING, (*Axis clearing state*)
		STATE_RESETTING (*Axis resetting state*)
		);
	ParameterStateEnum :
		(
		PAR_STATE_INIT, (*Param initialization state*)
		PAR_STATE_READ, (*Param read state*)
		PAR_STATE_WRITE, (*Param write state*)
		PAR_STATE_READY (*Param ready state*)
		);
	ConfigurationStateEnum :
		(
		CONFIG_STATE_INIT, (*Config initialization state*)
		CONFIG_STATE_READ, (*Config read state*)
		CONFIG_STATE_WRITE, (*Config write state*)
		CONFIG_STATE_READY (*Config ready state*)
		);
	ManualStateEnum :
		(
		MANUAL_STATE_IDLE, (*Idle state*)
		MANUAL_STATE_JOG, (*Jog state*)
		MANUAL_STATE_MOVE, (*Move state*)
		MANUAL_STATE_STOPPING (*Stopping state*)
		);
	AutomaticStateEnum :
		(
		AUTOMATIC_STATE_IDLE, (*Idle state*)
		AUTOMATIC_STATE_RUNNING (*Run state*)
		);
	AxisRecipeStepEnum :
		(
		REC_AXIS_WAIT, (*Wait state*)
		REC_AXIS_LOAD, (*Load product parameters*)
		REC_AXIS_SAVE, (*Save product parameters*)
		REC_AXIS_CREATE, (*Create new axis recipe*)
		REC_AXIS_STORE_MACH_SETTINGS, (*Save machine parameter settings*)
		REC_AXIS_FACTORY_RESET (*Factory reset*)
		);
END_TYPE
```

#### AxisMgr.var - not listed in the package file held
```iecst
VAR
	i : {REDUND_UNREPLICABLE} USINT; (*Loop index variable*)
	ParameterState : {REDUND_UNREPLICABLE} ParameterStateEnum; (*Parameter handling state*)
	ConfigurationState : {REDUND_UNREPLICABLE} ConfigurationStateEnum; (*Configuration handling state*)
	State : {REDUND_UNREPLICABLE} StateEnum; (*OMAC based state machine*)
	AutomaticState : {REDUND_UNREPLICABLE} AutomaticStateEnum; (*Automatic handling state*)
	ManualState : {REDUND_UNREPLICABLE} ManualStateEnum; (*Manual handling state*)
	AxisControl : {REDUND_UNREPLICABLE} AxisControlType := (Status:=(VisibilityControl:=[0,1])); (*Single axis control type*)
	AxisSettings : {REDUND_UNREPLICABLE} AxisSettingsType; (*Single axis settings *)
END_VAR
(*Function Blocks*)
VAR
	RestorePosition : {REDUND_UNREPLICABLE} McPureVAxRestorePosType; (*Data structure for retsore position mode*)
	MpRecipeRegPar_Cfg : {REDUND_UNREPLICABLE} MpRecipeRegPar; (*Register function block for configuration values*)
	MpRecipeRegPar_Par : {REDUND_UNREPLICABLE} MpRecipeRegPar; (*Register function block for parameter values*)
	MpAlarmXCore_0 : {REDUND_UNREPLICABLE} MpAlarmXCore; (*AlarmX Core function block*)
	MpAxisParameters : {REDUND_UNREPLICABLE} MpAxisBasicParType := (Distance:=70,Velocity:=100,Acceleration:=5000,Deceleration:=5000,Jog:=(Velocity:=70,Acceleration:=5000,Deceleration:=5000),AutoTune:=(MaxCurrentPercent:=50,MaxDistance:=720,MaxPositionError:=5)); (*Standard MpAxis parameter structure *)
	MpAxisBasic_0 : {REDUND_UNREPLICABLE} MpAxisBasic; (*MpAxis main function block*)
	MC_BR_ProcessConfig_AX : {REDUND_UNREPLICABLE} MC_BR_ProcessConfig; (*Function block to read and write the axis configuration*)
	MC_BR_ProcessConfig_ACP : {REDUND_UNREPLICABLE} MC_BR_ProcessConfig; (*Function block to read and write the ACOPOS configuration*)
	IsHomedEdgePos : {REDUND_UNREPLICABLE} R_TRIG; (*Detecting rising edge for Homed*)
	InPositionEdgePos : {REDUND_UNREPLICABLE} R_TRIG; (*Detecting rising edge for InPosition*)
	ReferenceEdgePos : {REDUND_UNREPLICABLE} R_TRIG; (*Detecting rising edge for Referenced*)
	MC_BR_ProcessParam_AX : {REDUND_UNREPLICABLE} MC_BR_ProcessParam; (*Function block to read and write the ACOPOS parameters*)
	MpAlarmXControl_SpeedNotSet : {REDUND_UNREPLICABLE} MpAlarmXAlarmControl; (*AlarmX control function block*)
END_VAR
(*Recipe*)
VAR
	ParametersEdit : {REDUND_UNREPLICABLE} AxisControlParametersType; (*Parameter structure used in recipe for edit*)
	ParametersPreview : {REDUND_UNREPLICABLE} AxisControlParametersType; (*Parameter structure used in recipe for preview*)
	MachineSettings : {REDUND_UNREPLICABLE} AxisMachineSettingsType; (*Machine settings structure*)
	MachineSettingsEdit : {REDUND_UNREPLICABLE} AxisMachineSettingsType; (*Machine settings structure used in recipe for edit*)
	MachineSettingsPreview : {REDUND_UNREPLICABLE} AxisMachineSettingsType; (*Machine settings structure used in recipe for preview*)
	AxisRecipe : {REDUND_UNREPLICABLE} AxisRecipeType; (*HMI interface structure*)
END_VAR
```

#### AxisStateMachine.st - not listed in the package file held
```iecst
ACTION AxisStateMachine:

	InPositionEdgePos.CLK := MpAxisBasic_0.InPosition;
	InPositionEdgePos();
	IsHomedEdgePos.CLK := MpAxisBasic_0.IsHomed;
	IsHomedEdgePos();
	ReferenceEdgePos.CLK := AxisControl.Command.Reference;
	ReferenceEdgePos();

	CASE State OF
		STATE_STOPPING..STATE_RESETTING:
			// Nothing to do as we are already handling any stop or errors in these states

		ELSE
			IF ((MpAxisBasic_0.Error = TRUE) OR MpAlarmXCheckReaction(gMpLinkAlarmXCore, 'Error')) THEN
				// Check alarm reaction
				ResetAllAxisCommands;
				State := STATE_ABORTING;
			ELSIF ((AxisControl.Command.Power = FALSE) AND (State > STATE_POWER_ON)) THEN
				ResetAllAxisCommands;
				AxisControl.Status.Busy := TRUE;
				MpAxisBasic_0.Power := FALSE;
				State := STATE_POWER_ON;
			END_IF

	END_CASE

	CASE State OF
		// Init state
		STATE_INIT:
			AxisControl.Status.Status := 'Initializing';
			ChangeConfiguration;
			ChangeParameter;
			IF ((ConfigurationState = CONFIG_STATE_READY) AND (ParameterState = PAR_STATE_READY) AND (MpAxisBasic_0.Active = TRUE)) THEN
				AxisControl.Status.IsReady := TRUE;

				State := STATE_POWER_ON;
			END_IF

		// Power on the axis
		STATE_POWER_ON:
			AxisControl.Status.Status := 'Waiting for power on';
			IF (MpAxisBasic_0.Info.ReadyToPowerOn = TRUE) THEN
				MpAxisBasic_0.Power := AxisControl.Command.Power;
			END_IF

			AxisControl.Status.Busy := MpAxisBasic_0.Power;
			IF (MpAxisBasic_0.PowerOn = TRUE) THEN
				AxisControl.Status.Busy := FALSE;
				State := STATE_HOME;
			ELSE
				ChangeConfiguration;
			END_IF

		// Restore home position
		STATE_HOME:
			AxisControl.Status.Status := 'Waiting for home';
			IF ((MpAxisBasic_0.IsHomed = FALSE) AND (MpAxisBasic_0.PowerOn = TRUE)) THEN
				AxisControl.Status.ReferenceRequired := TRUE;
				State := STATE_REFERENCE;
			END_IF

			IF (MpAxisBasic_0.IsHomed = TRUE) THEN
				AxisControl.Status.ReferenceRequired := FALSE;
				AxisControl.Status.Busy := FALSE;
				AxisControl.Command.Reference := FALSE;
				State := STATE_MOVE_TO_HOME_POSITION;
				ResetAllAxisCommands;
			END_IF

		// Create reference position
		STATE_REFERENCE:
			IF (AxisControl.Command.Reference = TRUE) THEN
				AxisControl.Command.Reference := FALSE;
				MpAxisBasic_0.Home := TRUE;
				AxisControl.Status.Busy := TRUE;
				MpAxisParameters.Homing.Mode := mcHOMING_DIRECT;
				MpAxisParameters.Homing.Position := MachineSettings.ReferencePosition;
			END_IF

			IF (IsHomedEdgePos.Q	= TRUE) THEN
				AxisControl.Status.ReferenceRequired := FALSE;
				State := STATE_MOVE_TO_HOME_POSITION;
				ResetAllAxisCommands;
			END_IF

		// Move to home position
		STATE_MOVE_TO_HOME_POSITION:
			AxisControl.Status.Status := 'Moving to home position';
			MpAxisParameters.Position := AxisControl.Parameters.HomePosition;
			MpAxisParameters.Direction := mcDIR_SHORTEST_WAY;
			MpAxisBasic_0.MoveAbsolute := TRUE;
			IF (InPositionEdgePos.Q	= TRUE) THEN
				AxisControl.Status.Busy := FALSE;
				MpAxisBasic_0.MoveAbsolute := FALSE;
				MpAxisParameters.Direction := mcDIR_POSITIVE;
				State := STATE_READY;
			END_IF

		// In this State the module is error free and ready for a command (manual or automatic)
		STATE_READY:
			AxisControl.Status.Status := 'Ready';
			AxisControl.Status.Busy := FALSE;
			IF (ReferenceEdgePos.Q = TRUE) THEN
				State := STATE_REFERENCE;
			ELSIF ((MpAlarmXCheckReaction(gMpLinkAlarmXCore, 'Warning') = FALSE) AND (AutomaticCommand(AxisControl.Command) = TRUE)) THEN
				State := STATE_AUTOMATIC_OPERATION;
			ELSIF (ManualCommand(AxisControl.Command) = TRUE) THEN
				State := STATE_MANUAL_OPERATION;
			END_IF

		// Axis can be moved manually / jogged
		STATE_MANUAL_OPERATION:
			AxisControl.Status.Status := 'Manual running';
			AxisControl.Status.Busy := TRUE;
			AxisManual;

		// Axis put into automatic mode / camming
		STATE_AUTOMATIC_OPERATION:
			AxisControl.Status.Status := 'Automatic running';
			AxisControl.Status.Busy := TRUE;
			IF MpAlarmXCheckReaction(gMpLinkAlarmXCore, 'Error') THEN
				AxisControl.Command.Stop := TRUE;
			END_IF

			AxisAutomatic;

		// In this State the module will attempt to bring the axis to a controlled stop.
		STATE_STOPPING:
			AxisControl.Status.Status := 'Stopping';

			// Stop the axis if it is powered on
			MpAxisBasic_0.Stop := MpAxisBasic_0.PowerOn;
			MpAxisParameters.Stop.Deceleration := AxisControl.Parameters.StopDeceleration;
			IF ((MpAxisBasic_0.PowerOn = FALSE) OR (MpAxisBasic_0.Stopped = TRUE)) THEN
				MpAxisBasic_0.Stop := FALSE;
				State := STATE_STOPPED;
			END_IF

		// In this State the module is powered on and at standstill.
		STATE_STOPPED:
			State := STATE_RESETTING;

		// In this State the module will bring the axis to a rapid stop
		STATE_ABORTING:
			MpAxisParameters.Stop.Deceleration := 0;
			MpAxisBasic_0.Stop := MpAxisBasic_0.PowerOn;
			IF ((MpAxisBasic_0.PowerOn = FALSE) OR (MpAxisBasic_0.Stopped = TRUE)) THEN
				MpAxisBasic_0.Stop := FALSE;
				IF (MpAlarmXCheckReaction(gMpLinkAlarmXCore, 'SafetyError') = TRUE) THEN
					// Safety errors also power off the axis
					MpAxisBasic_0.Power := FALSE;
					IF (MpAxisBasic_0.PowerOn = FALSE) THEN
						State := STATE_ABORTED;
					END_IF
				ELSE
					State := STATE_ABORTED;
				END_IF
			END_IF

		STATE_ABORTED:
			State := STATE_CLEARING;

		STATE_CLEARING:
			State := STATE_RESETTING;

		// In this State the module attempts to clear any outstanding errors.  No hazardous motion should occur in this State.
		STATE_RESETTING:
			ResetAllAxisCommands;
			IF (AxisControl.Command.Reset = TRUE) OR ((MpAlarmXCheckReaction(gMpLinkAlarmXCore, 'Error') = FALSE) AND EDGEPOS(MpAlarmXCore_0.PendingAlarms = 0)) THEN
				AxisControl.Status.Busy := TRUE;
				AxisControl.Command.Reset := FALSE;
				MpAxisBasic_0.ErrorReset := TRUE;
				AxisReset;
				ManualState := MANUAL_STATE_IDLE;
				AutomaticState := AUTOMATIC_STATE_IDLE;
			ELSE
				MpAxisBasic_0.ErrorReset := FALSE;
			END_IF

			IF ((MpAxisBasic_0.Error = FALSE) AND (MpAlarmXCheckReaction(gMpLinkAlarmXCore, 'Error') = FALSE)) THEN
				AxisControl.Status.Busy := FALSE;
				IF (MpAxisBasic_0.PowerOn = FALSE) THEN
					State := STATE_POWER_ON;
				ELSIF (MpAxisBasic_0.IsHomed = TRUE) THEN
					State := STATE_READY;
				ELSE
					State := STATE_HOME;
				END_IF
			END_IF

	END_CASE

	// Cyclic function block calls
	MpAxisBasic_0.Parameters := ADR(MpAxisParameters);
	MpAxisBasic_0();

	// Status assignments
	AxisControl.Status.ErrorActive := MpAxisBasic_0.Error OR (MpAlarmXCheckReaction(gMpLinkAlarmXCore, 'Error'));
	AxisControl.Status.IsHomed := MpAxisBasic_0.IsHomed;
	AxisControl.Status.IsPowered := MpAxisBasic_0.PowerOn;
	AxisControl.Status.PLCopenState := MpAxisBasic_0.Info.PLCopenState;
	AxisControl.Status.Position := MpAxisBasic_0.Position;
	AxisControl.Status.Velocity := MpAxisBasic_0.Velocity;
	AxisControl.Status.ModeManual := (State <> STATE_AUTOMATIC_OPERATION);
	//VC4 related code
	AxisControl.Status.StatusPointControl[0].0 := NOT AxisControl.Status.StatusPointControl[1].0;
	AxisControl.Status.StatusPointControl[0].1 := NOT AxisControl.Status.ModeManual;

END_ACTION

ACTION ResetAllAxisCommands:

	MpAxisBasic_0.MoveAbsolute := FALSE;
	MpAxisBasic_0.MoveAdditive := FALSE;
	MpAxisBasic_0.MoveVelocity := FALSE;
	MpAxisBasic_0.ReleaseBrake := FALSE;
	MpAxisBasic_0.ErrorReset := FALSE;
	MpAxisBasic_0.JogPositive := FALSE;
	MpAxisBasic_0.JogNegative := FALSE;
	MpAxisBasic_0.Home := FALSE;

END_ACTION
```

#### ChangeConfiguration.st - not listed in the package file held
```iecst
ACTION ConfigurationInit:
	// Initalize drive configuration
	AxisSettings.DriveConfiguration.PureVirtualAxis.AxisFeatures.FeatureReference.DataAddress := ADR(AxisSettings.AxisFeatures);
	AxisSettings.DriveConfiguration.PureVirtualAxis.AxisFeatures.FeatureReference.NumberOfArrayElements := SIZEOF(AxisSettings.AxisFeatures)/SIZEOF(AxisSettings.AxisFeatures[0]);
	AxisSettings.DriveConfiguration.PureVirtualAxis.AxisFeatures.FeatureReference.NumberOfElements := 0;
	i := 0;
	WHILE ((i <= SIZEOF(AxisSettings.AxisFeatures)/SIZEOF(AxisSettings.AxisFeatures[0])) AND (AxisSettings.AxisFeatures[i] <> '')) DO
		i := i + 1;
	END_WHILE
	AxisSettings.DriveConfiguration.PureVirtualAxis.AxisFeatures.FeatureReference.NumberOfElements := i;

	MC_BR_ProcessConfig_AX.DataAddress := ADR(AxisSettings.BaseConfiguration);
	MC_BR_ProcessConfig_AX.DataType := mcCFG_AX;

	MC_BR_ProcessConfig_ACP.DataAddress := ADR(AxisSettings.DriveConfiguration);
	MC_BR_ProcessConfig_ACP.DataType := mcCFG_PURE_V_AX;

	ConfigurationState := CONFIG_STATE_INIT;

END_ACTION

ACTION ChangeConfiguration:

	CASE ConfigurationState OF
		CONFIG_STATE_INIT:

			// Assign string for the name
			MC_BR_ProcessConfig_ACP.Name := MpAxisBasic_0.Info.HardwareInfo.Axis.ConfigElementLocation;
			MC_BR_ProcessConfig_AX.Name := MpAxisBasic_0.Info.HardwareInfo.Axis.AxisName;

			IF (MpAxisBasic_0.Active = TRUE) THEN
				ConfigurationState := CONFIG_STATE_READ;
			END_IF

		CONFIG_STATE_READ:
			// Read the current configuration
			MC_BR_ProcessConfig_ACP.Mode := mcPCM_LOAD;
			MC_BR_ProcessConfig_ACP.Execute := TRUE;

			MC_BR_ProcessConfig_AX.Mode := mcPCM_LOAD;
			MC_BR_ProcessConfig_AX.Execute := TRUE;
			IF (MC_BR_ProcessConfig_ACP.Done = TRUE) AND (MC_BR_ProcessConfig_AX.Done = TRUE) THEN
				MC_BR_ProcessConfig_ACP.Execute := FALSE;
				MC_BR_ProcessConfig_AX.Execute := FALSE;
				ConfigurationState := CONFIG_STATE_READY;
			END_IF

		CONFIG_STATE_WRITE:
			// Write the configuration after changes
			MC_BR_ProcessConfig_ACP.Mode := mcPCM_SAVE;
			MC_BR_ProcessConfig_ACP.Execute := TRUE;

			MC_BR_ProcessConfig_AX.Mode := mcPCM_SAVE;
			MC_BR_ProcessConfig_AX.Execute := TRUE;
			IF (MC_BR_ProcessConfig_ACP.Done = TRUE) AND (MC_BR_ProcessConfig_AX.Done = TRUE) THEN
				MC_BR_ProcessConfig_ACP.Execute := FALSE;
				MC_BR_ProcessConfig_AX.Execute := FALSE;
				ConfigurationState := CONFIG_STATE_READY;
			END_IF

		CONFIG_STATE_READY:

	END_CASE

	// Cyclic function block calls
	AxisSettings.DriveConfiguration.PureVirtualAxis.AxisFeatures.FeatureReference.DataAddress := ADR(AxisSettings.AxisFeatures);
	MC_BR_ProcessConfig_AX.DataAddress := ADR(AxisSettings.BaseConfiguration);
	MC_BR_ProcessConfig_ACP.DataAddress := ADR(AxisSettings.DriveConfiguration);
	MC_BR_ProcessConfig_ACP();
	MC_BR_ProcessConfig_AX();

END_ACTION

ACTION ParameterInit:
	// Initalize drive parameter
	MC_BR_ProcessParam_AX.DataAddress := ADR(AxisSettings.BaseParam);
	MC_BR_ProcessParam_AX.DataType := mcCFG_AX_MOVE_LIM;

	ParameterState := PAR_STATE_INIT;

END_ACTION

ACTION ChangeParameter:

	CASE ParameterState OF
		PAR_STATE_INIT:
			// Wait state
			MC_BR_ProcessParam_AX.Component := MpAxisBasic_0.MpLink;

			IF (MpAxisBasic_0.Active = TRUE) THEN
				ParameterState := PAR_STATE_READ;
			END_IF

		PAR_STATE_READ:
			// Read current parameter values
			MC_BR_ProcessParam_AX.Mode := mcPPM_READ;
			MC_BR_ProcessParam_AX.Execute := TRUE;

			IF (MC_BR_ProcessParam_AX.Done = TRUE) THEN
				MC_BR_ProcessParam_AX.Execute := FALSE;
				ParameterState := PAR_STATE_READY;
			END_IF

		PAR_STATE_WRITE:
			// Write new parameter values
			MC_BR_ProcessParam_AX.Mode := mcPPM_WRITE;
			MC_BR_ProcessParam_AX.Execute := TRUE;

			IF (MC_BR_ProcessParam_AX.Done = TRUE) THEN
				MC_BR_ProcessParam_AX.Execute := FALSE;
				ParameterState := PAR_STATE_READY;
			END_IF

		PAR_STATE_READY:

	END_CASE

	MC_BR_ProcessParam_AX.DataAddress := ADR(AxisSettings.BaseParam);
	MC_BR_ProcessParam_AX();

END_ACTION
```
